// TIA Portal V18 export
FUNCTION "SS2_A3_32DI_IO_Update" : Void   // FC11140, LAD
{ S7_Optimized_Access := 'TRUE' }
VERSION : 0.1
// stored: AutoNumber false, IsIECCheckEnabled false, SetENOAutomatically false, UDAEnableTagReadback false
BEGIN

REGION Network 1: DIa0
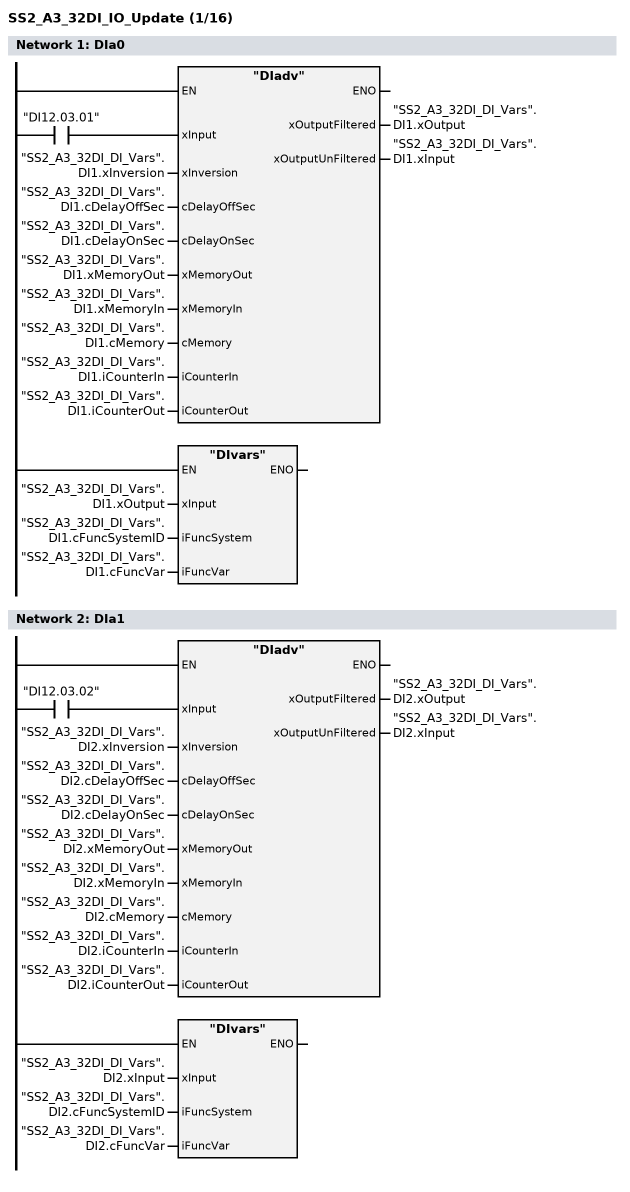
   RUNG wire#powerrail
      "DIadv"(xInput := wire#w1, xInversion := "SS2_A3_32DI_DI_Vars".DI1.xInversion, cDelayOffSec := "SS2_A3_32DI_DI_Vars".DI1.cDelayOffSec, cDelayOnSec := "SS2_A3_32DI_DI_Vars".DI1.cDelayOnSec, xMemoryOut := "SS2_A3_32DI_DI_Vars".DI1.xMemoryOut, xMemoryIn := "SS2_A3_32DI_DI_Vars".DI1.xMemoryIn, cMemory := "SS2_A3_32DI_DI_Vars".DI1.cMemory, iCounterIn := "SS2_A3_32DI_DI_Vars".DI1.iCounterIn, iCounterOut := "SS2_A3_32DI_DI_Vars".DI1.iCounterOut, xOutputFiltered => "SS2_A3_32DI_DI_Vars".DI1.xOutput, xOutputUnFiltered => "SS2_A3_32DI_DI_Vars".DI1.xInput)
   END_RUNG
   RUNG wire#powerrail
      Contact( "DI12.03.01" )
   END_RUNG wire#w1
   RUNG wire#powerrail
      "DIvars"(xInput := "SS2_A3_32DI_DI_Vars".DI1.xOutput, iFuncSystem := "SS2_A3_32DI_DI_Vars".DI1.cFuncSystemID, iFuncVar := "SS2_A3_32DI_DI_Vars".DI1.cFuncVar)
   END_RUNG
   // the same network as SCL:
   "DIadv"(xInput := "DI12.03.01",
           xInversion := "SS2_A3_32DI_DI_Vars".DI1.xInversion,
           cDelayOffSec := "SS2_A3_32DI_DI_Vars".DI1.cDelayOffSec,
           cDelayOnSec := "SS2_A3_32DI_DI_Vars".DI1.cDelayOnSec,
           xMemoryOut := "SS2_A3_32DI_DI_Vars".DI1.xMemoryOut,
           xMemoryIn := "SS2_A3_32DI_DI_Vars".DI1.xMemoryIn,
           cMemory := "SS2_A3_32DI_DI_Vars".DI1.cMemory,
           iCounterIn := "SS2_A3_32DI_DI_Vars".DI1.iCounterIn,
           iCounterOut := "SS2_A3_32DI_DI_Vars".DI1.iCounterOut,
           xOutputFiltered => "SS2_A3_32DI_DI_Vars".DI1.xOutput,
           xOutputUnFiltered => "SS2_A3_32DI_DI_Vars".DI1.xInput);
   "DIvars"(xInput := "SS2_A3_32DI_DI_Vars".DI1.xOutput,
            iFuncSystem := "SS2_A3_32DI_DI_Vars".DI1.cFuncSystemID,
            iFuncVar := "SS2_A3_32DI_DI_Vars".DI1.cFuncVar);
END_REGION

REGION Network 2: DIa1
   RUNG wire#powerrail
      "DIadv"(xInput := wire#w1, xInversion := "SS2_A3_32DI_DI_Vars".DI2.xInversion, cDelayOffSec := "SS2_A3_32DI_DI_Vars".DI2.cDelayOffSec, cDelayOnSec := "SS2_A3_32DI_DI_Vars".DI2.cDelayOnSec, xMemoryOut := "SS2_A3_32DI_DI_Vars".DI2.xMemoryOut, xMemoryIn := "SS2_A3_32DI_DI_Vars".DI2.xMemoryIn, cMemory := "SS2_A3_32DI_DI_Vars".DI2.cMemory, iCounterIn := "SS2_A3_32DI_DI_Vars".DI2.iCounterIn, iCounterOut := "SS2_A3_32DI_DI_Vars".DI2.iCounterOut, xOutputFiltered => "SS2_A3_32DI_DI_Vars".DI2.xOutput, xOutputUnFiltered => "SS2_A3_32DI_DI_Vars".DI2.xInput)
   END_RUNG
   RUNG wire#powerrail
      Contact( "DI12.03.02" )
   END_RUNG wire#w1
   RUNG wire#powerrail
      "DIvars"(xInput := "SS2_A3_32DI_DI_Vars".DI2.xInput, iFuncSystem := "SS2_A3_32DI_DI_Vars".DI2.cFuncSystemID, iFuncVar := "SS2_A3_32DI_DI_Vars".DI2.cFuncVar)
   END_RUNG
   // the same network as SCL:
   "DIadv"(xInput := "DI12.03.02",
           xInversion := "SS2_A3_32DI_DI_Vars".DI2.xInversion,
           cDelayOffSec := "SS2_A3_32DI_DI_Vars".DI2.cDelayOffSec,
           cDelayOnSec := "SS2_A3_32DI_DI_Vars".DI2.cDelayOnSec,
           xMemoryOut := "SS2_A3_32DI_DI_Vars".DI2.xMemoryOut,
           xMemoryIn := "SS2_A3_32DI_DI_Vars".DI2.xMemoryIn,
           cMemory := "SS2_A3_32DI_DI_Vars".DI2.cMemory,
           iCounterIn := "SS2_A3_32DI_DI_Vars".DI2.iCounterIn,
           iCounterOut := "SS2_A3_32DI_DI_Vars".DI2.iCounterOut,
           xOutputFiltered => "SS2_A3_32DI_DI_Vars".DI2.xOutput,
           xOutputUnFiltered => "SS2_A3_32DI_DI_Vars".DI2.xInput);
   "DIvars"(xInput := "SS2_A3_32DI_DI_Vars".DI2.xInput,
            iFuncSystem := "SS2_A3_32DI_DI_Vars".DI2.cFuncSystemID,
            iFuncVar := "SS2_A3_32DI_DI_Vars".DI2.cFuncVar);
END_REGION

REGION Network 3: DIa2
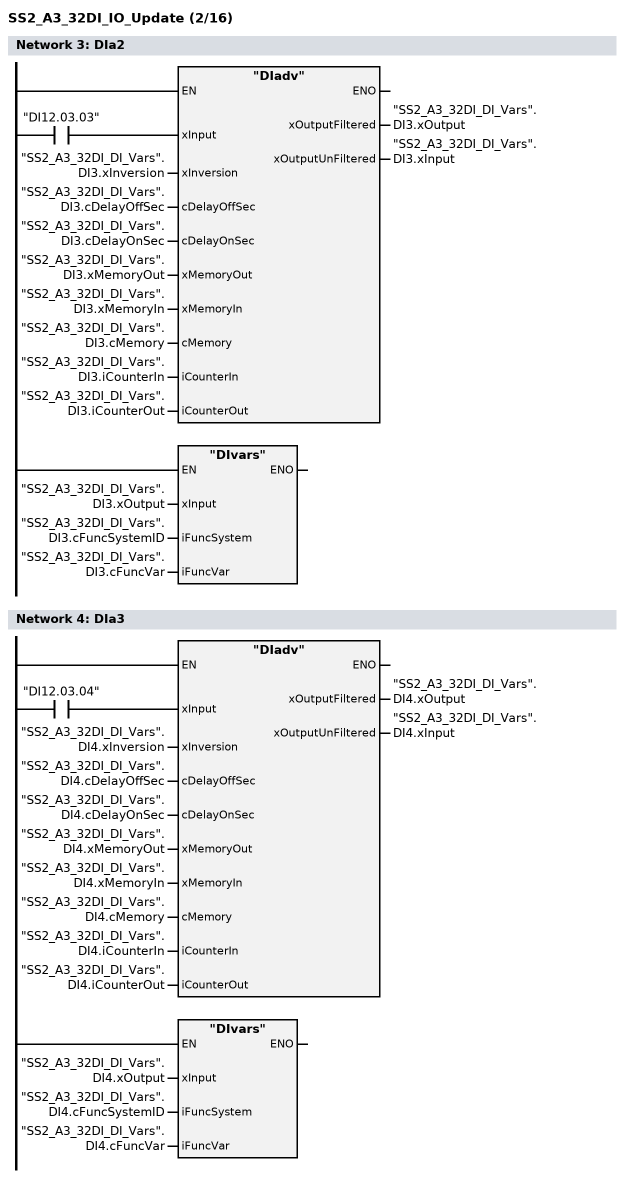
   RUNG wire#powerrail
      "DIadv"(xInput := wire#w1, xInversion := "SS2_A3_32DI_DI_Vars".DI3.xInversion, cDelayOffSec := "SS2_A3_32DI_DI_Vars".DI3.cDelayOffSec, cDelayOnSec := "SS2_A3_32DI_DI_Vars".DI3.cDelayOnSec, xMemoryOut := "SS2_A3_32DI_DI_Vars".DI3.xMemoryOut, xMemoryIn := "SS2_A3_32DI_DI_Vars".DI3.xMemoryIn, cMemory := "SS2_A3_32DI_DI_Vars".DI3.cMemory, iCounterIn := "SS2_A3_32DI_DI_Vars".DI3.iCounterIn, iCounterOut := "SS2_A3_32DI_DI_Vars".DI3.iCounterOut, xOutputFiltered => "SS2_A3_32DI_DI_Vars".DI3.xOutput, xOutputUnFiltered => "SS2_A3_32DI_DI_Vars".DI3.xInput)
   END_RUNG
   RUNG wire#powerrail
      Contact( "DI12.03.03" )
   END_RUNG wire#w1
   RUNG wire#powerrail
      "DIvars"(xInput := "SS2_A3_32DI_DI_Vars".DI3.xOutput, iFuncSystem := "SS2_A3_32DI_DI_Vars".DI3.cFuncSystemID, iFuncVar := "SS2_A3_32DI_DI_Vars".DI3.cFuncVar)
   END_RUNG
   // the same network as SCL:
   "DIadv"(xInput := "DI12.03.03",
           xInversion := "SS2_A3_32DI_DI_Vars".DI3.xInversion,
           cDelayOffSec := "SS2_A3_32DI_DI_Vars".DI3.cDelayOffSec,
           cDelayOnSec := "SS2_A3_32DI_DI_Vars".DI3.cDelayOnSec,
           xMemoryOut := "SS2_A3_32DI_DI_Vars".DI3.xMemoryOut,
           xMemoryIn := "SS2_A3_32DI_DI_Vars".DI3.xMemoryIn,
           cMemory := "SS2_A3_32DI_DI_Vars".DI3.cMemory,
           iCounterIn := "SS2_A3_32DI_DI_Vars".DI3.iCounterIn,
           iCounterOut := "SS2_A3_32DI_DI_Vars".DI3.iCounterOut,
           xOutputFiltered => "SS2_A3_32DI_DI_Vars".DI3.xOutput,
           xOutputUnFiltered => "SS2_A3_32DI_DI_Vars".DI3.xInput);
   "DIvars"(xInput := "SS2_A3_32DI_DI_Vars".DI3.xOutput,
            iFuncSystem := "SS2_A3_32DI_DI_Vars".DI3.cFuncSystemID,
            iFuncVar := "SS2_A3_32DI_DI_Vars".DI3.cFuncVar);
END_REGION

REGION Network 4: DIa3
   RUNG wire#powerrail
      "DIadv"(xInput := wire#w1, xInversion := "SS2_A3_32DI_DI_Vars".DI4.xInversion, cDelayOffSec := "SS2_A3_32DI_DI_Vars".DI4.cDelayOffSec, cDelayOnSec := "SS2_A3_32DI_DI_Vars".DI4.cDelayOnSec, xMemoryOut := "SS2_A3_32DI_DI_Vars".DI4.xMemoryOut, xMemoryIn := "SS2_A3_32DI_DI_Vars".DI4.xMemoryIn, cMemory := "SS2_A3_32DI_DI_Vars".DI4.cMemory, iCounterIn := "SS2_A3_32DI_DI_Vars".DI4.iCounterIn, iCounterOut := "SS2_A3_32DI_DI_Vars".DI4.iCounterOut, xOutputFiltered => "SS2_A3_32DI_DI_Vars".DI4.xOutput, xOutputUnFiltered => "SS2_A3_32DI_DI_Vars".DI4.xInput)
   END_RUNG
   RUNG wire#powerrail
      Contact( "DI12.03.04" )
   END_RUNG wire#w1
   RUNG wire#powerrail
      "DIvars"(xInput := "SS2_A3_32DI_DI_Vars".DI4.xOutput, iFuncSystem := "SS2_A3_32DI_DI_Vars".DI4.cFuncSystemID, iFuncVar := "SS2_A3_32DI_DI_Vars".DI4.cFuncVar)
   END_RUNG
   // the same network as SCL:
   "DIadv"(xInput := "DI12.03.04",
           xInversion := "SS2_A3_32DI_DI_Vars".DI4.xInversion,
           cDelayOffSec := "SS2_A3_32DI_DI_Vars".DI4.cDelayOffSec,
           cDelayOnSec := "SS2_A3_32DI_DI_Vars".DI4.cDelayOnSec,
           xMemoryOut := "SS2_A3_32DI_DI_Vars".DI4.xMemoryOut,
           xMemoryIn := "SS2_A3_32DI_DI_Vars".DI4.xMemoryIn,
           cMemory := "SS2_A3_32DI_DI_Vars".DI4.cMemory,
           iCounterIn := "SS2_A3_32DI_DI_Vars".DI4.iCounterIn,
           iCounterOut := "SS2_A3_32DI_DI_Vars".DI4.iCounterOut,
           xOutputFiltered => "SS2_A3_32DI_DI_Vars".DI4.xOutput,
           xOutputUnFiltered => "SS2_A3_32DI_DI_Vars".DI4.xInput);
   "DIvars"(xInput := "SS2_A3_32DI_DI_Vars".DI4.xOutput,
            iFuncSystem := "SS2_A3_32DI_DI_Vars".DI4.cFuncSystemID,
            iFuncVar := "SS2_A3_32DI_DI_Vars".DI4.cFuncVar);
END_REGION

REGION Network 5: DIa4
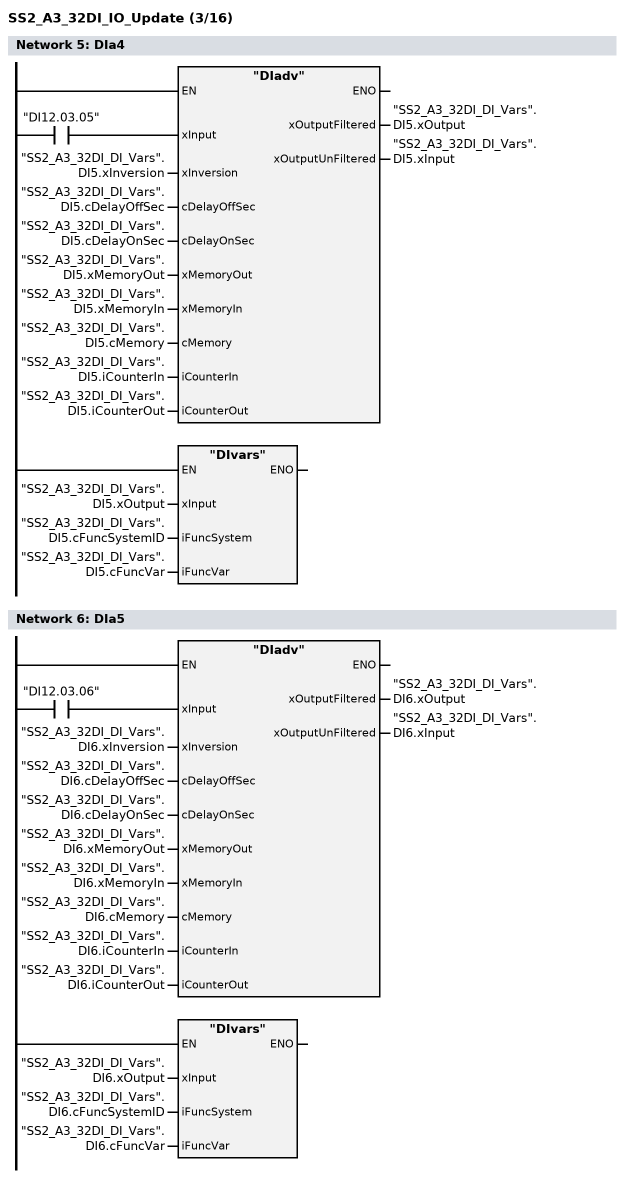
   RUNG wire#powerrail
      "DIadv"(xInput := wire#w1, xInversion := "SS2_A3_32DI_DI_Vars".DI5.xInversion, cDelayOffSec := "SS2_A3_32DI_DI_Vars".DI5.cDelayOffSec, cDelayOnSec := "SS2_A3_32DI_DI_Vars".DI5.cDelayOnSec, xMemoryOut := "SS2_A3_32DI_DI_Vars".DI5.xMemoryOut, xMemoryIn := "SS2_A3_32DI_DI_Vars".DI5.xMemoryIn, cMemory := "SS2_A3_32DI_DI_Vars".DI5.cMemory, iCounterIn := "SS2_A3_32DI_DI_Vars".DI5.iCounterIn, iCounterOut := "SS2_A3_32DI_DI_Vars".DI5.iCounterOut, xOutputFiltered => "SS2_A3_32DI_DI_Vars".DI5.xOutput, xOutputUnFiltered => "SS2_A3_32DI_DI_Vars".DI5.xInput)
   END_RUNG
   RUNG wire#powerrail
      Contact( "DI12.03.05" )
   END_RUNG wire#w1
   RUNG wire#powerrail
      "DIvars"(xInput := "SS2_A3_32DI_DI_Vars".DI5.xOutput, iFuncSystem := "SS2_A3_32DI_DI_Vars".DI5.cFuncSystemID, iFuncVar := "SS2_A3_32DI_DI_Vars".DI5.cFuncVar)
   END_RUNG
   // the same network as SCL:
   "DIadv"(xInput := "DI12.03.05",
           xInversion := "SS2_A3_32DI_DI_Vars".DI5.xInversion,
           cDelayOffSec := "SS2_A3_32DI_DI_Vars".DI5.cDelayOffSec,
           cDelayOnSec := "SS2_A3_32DI_DI_Vars".DI5.cDelayOnSec,
           xMemoryOut := "SS2_A3_32DI_DI_Vars".DI5.xMemoryOut,
           xMemoryIn := "SS2_A3_32DI_DI_Vars".DI5.xMemoryIn,
           cMemory := "SS2_A3_32DI_DI_Vars".DI5.cMemory,
           iCounterIn := "SS2_A3_32DI_DI_Vars".DI5.iCounterIn,
           iCounterOut := "SS2_A3_32DI_DI_Vars".DI5.iCounterOut,
           xOutputFiltered => "SS2_A3_32DI_DI_Vars".DI5.xOutput,
           xOutputUnFiltered => "SS2_A3_32DI_DI_Vars".DI5.xInput);
   "DIvars"(xInput := "SS2_A3_32DI_DI_Vars".DI5.xOutput,
            iFuncSystem := "SS2_A3_32DI_DI_Vars".DI5.cFuncSystemID,
            iFuncVar := "SS2_A3_32DI_DI_Vars".DI5.cFuncVar);
END_REGION

REGION Network 6: DIa5
   RUNG wire#powerrail
      "DIadv"(xInput := wire#w1, xInversion := "SS2_A3_32DI_DI_Vars".DI6.xInversion, cDelayOffSec := "SS2_A3_32DI_DI_Vars".DI6.cDelayOffSec, cDelayOnSec := "SS2_A3_32DI_DI_Vars".DI6.cDelayOnSec, xMemoryOut := "SS2_A3_32DI_DI_Vars".DI6.xMemoryOut, xMemoryIn := "SS2_A3_32DI_DI_Vars".DI6.xMemoryIn, cMemory := "SS2_A3_32DI_DI_Vars".DI6.cMemory, iCounterIn := "SS2_A3_32DI_DI_Vars".DI6.iCounterIn, iCounterOut := "SS2_A3_32DI_DI_Vars".DI6.iCounterOut, xOutputFiltered => "SS2_A3_32DI_DI_Vars".DI6.xOutput, xOutputUnFiltered => "SS2_A3_32DI_DI_Vars".DI6.xInput)
   END_RUNG
   RUNG wire#powerrail
      Contact( "DI12.03.06" )
   END_RUNG wire#w1
   RUNG wire#powerrail
      "DIvars"(xInput := "SS2_A3_32DI_DI_Vars".DI6.xOutput, iFuncSystem := "SS2_A3_32DI_DI_Vars".DI6.cFuncSystemID, iFuncVar := "SS2_A3_32DI_DI_Vars".DI6.cFuncVar)
   END_RUNG
   // the same network as SCL:
   "DIadv"(xInput := "DI12.03.06",
           xInversion := "SS2_A3_32DI_DI_Vars".DI6.xInversion,
           cDelayOffSec := "SS2_A3_32DI_DI_Vars".DI6.cDelayOffSec,
           cDelayOnSec := "SS2_A3_32DI_DI_Vars".DI6.cDelayOnSec,
           xMemoryOut := "SS2_A3_32DI_DI_Vars".DI6.xMemoryOut,
           xMemoryIn := "SS2_A3_32DI_DI_Vars".DI6.xMemoryIn,
           cMemory := "SS2_A3_32DI_DI_Vars".DI6.cMemory,
           iCounterIn := "SS2_A3_32DI_DI_Vars".DI6.iCounterIn,
           iCounterOut := "SS2_A3_32DI_DI_Vars".DI6.iCounterOut,
           xOutputFiltered => "SS2_A3_32DI_DI_Vars".DI6.xOutput,
           xOutputUnFiltered => "SS2_A3_32DI_DI_Vars".DI6.xInput);
   "DIvars"(xInput := "SS2_A3_32DI_DI_Vars".DI6.xOutput,
            iFuncSystem := "SS2_A3_32DI_DI_Vars".DI6.cFuncSystemID,
            iFuncVar := "SS2_A3_32DI_DI_Vars".DI6.cFuncVar);
END_REGION

REGION Network 7: DIa6
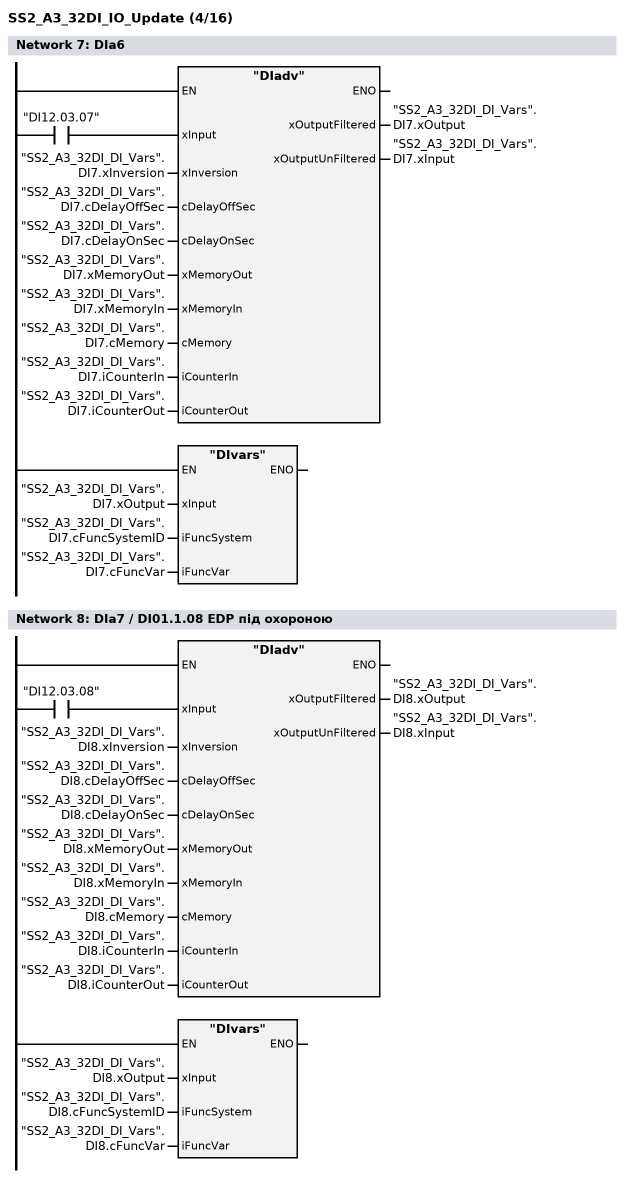
   RUNG wire#powerrail
      "DIadv"(xInput := wire#w1, xInversion := "SS2_A3_32DI_DI_Vars".DI7.xInversion, cDelayOffSec := "SS2_A3_32DI_DI_Vars".DI7.cDelayOffSec, cDelayOnSec := "SS2_A3_32DI_DI_Vars".DI7.cDelayOnSec, xMemoryOut := "SS2_A3_32DI_DI_Vars".DI7.xMemoryOut, xMemoryIn := "SS2_A3_32DI_DI_Vars".DI7.xMemoryIn, cMemory := "SS2_A3_32DI_DI_Vars".DI7.cMemory, iCounterIn := "SS2_A3_32DI_DI_Vars".DI7.iCounterIn, iCounterOut := "SS2_A3_32DI_DI_Vars".DI7.iCounterOut, xOutputFiltered => "SS2_A3_32DI_DI_Vars".DI7.xOutput, xOutputUnFiltered => "SS2_A3_32DI_DI_Vars".DI7.xInput)
   END_RUNG
   RUNG wire#powerrail
      Contact( "DI12.03.07" )
   END_RUNG wire#w1
   RUNG wire#powerrail
      "DIvars"(xInput := "SS2_A3_32DI_DI_Vars".DI7.xOutput, iFuncSystem := "SS2_A3_32DI_DI_Vars".DI7.cFuncSystemID, iFuncVar := "SS2_A3_32DI_DI_Vars".DI7.cFuncVar)
   END_RUNG
   // the same network as SCL:
   "DIadv"(xInput := "DI12.03.07",
           xInversion := "SS2_A3_32DI_DI_Vars".DI7.xInversion,
           cDelayOffSec := "SS2_A3_32DI_DI_Vars".DI7.cDelayOffSec,
           cDelayOnSec := "SS2_A3_32DI_DI_Vars".DI7.cDelayOnSec,
           xMemoryOut := "SS2_A3_32DI_DI_Vars".DI7.xMemoryOut,
           xMemoryIn := "SS2_A3_32DI_DI_Vars".DI7.xMemoryIn,
           cMemory := "SS2_A3_32DI_DI_Vars".DI7.cMemory,
           iCounterIn := "SS2_A3_32DI_DI_Vars".DI7.iCounterIn,
           iCounterOut := "SS2_A3_32DI_DI_Vars".DI7.iCounterOut,
           xOutputFiltered => "SS2_A3_32DI_DI_Vars".DI7.xOutput,
           xOutputUnFiltered => "SS2_A3_32DI_DI_Vars".DI7.xInput);
   "DIvars"(xInput := "SS2_A3_32DI_DI_Vars".DI7.xOutput,
            iFuncSystem := "SS2_A3_32DI_DI_Vars".DI7.cFuncSystemID,
            iFuncVar := "SS2_A3_32DI_DI_Vars".DI7.cFuncVar);
END_REGION

REGION Network 8: DIa7 / DI01.1.08 EDP під охороною
   RUNG wire#powerrail
      "DIadv"(xInput := wire#w1, xInversion := "SS2_A3_32DI_DI_Vars".DI8.xInversion, cDelayOffSec := "SS2_A3_32DI_DI_Vars".DI8.cDelayOffSec, cDelayOnSec := "SS2_A3_32DI_DI_Vars".DI8.cDelayOnSec, xMemoryOut := "SS2_A3_32DI_DI_Vars".DI8.xMemoryOut, xMemoryIn := "SS2_A3_32DI_DI_Vars".DI8.xMemoryIn, cMemory := "SS2_A3_32DI_DI_Vars".DI8.cMemory, iCounterIn := "SS2_A3_32DI_DI_Vars".DI8.iCounterIn, iCounterOut := "SS2_A3_32DI_DI_Vars".DI8.iCounterOut, xOutputFiltered => "SS2_A3_32DI_DI_Vars".DI8.xOutput, xOutputUnFiltered => "SS2_A3_32DI_DI_Vars".DI8.xInput)
   END_RUNG
   RUNG wire#powerrail
      Contact( "DI12.03.08" )
   END_RUNG wire#w1
   RUNG wire#powerrail
      "DIvars"(xInput := "SS2_A3_32DI_DI_Vars".DI8.xOutput, iFuncSystem := "SS2_A3_32DI_DI_Vars".DI8.cFuncSystemID, iFuncVar := "SS2_A3_32DI_DI_Vars".DI8.cFuncVar)
   END_RUNG
   // the same network as SCL:
   "DIadv"(xInput := "DI12.03.08",
           xInversion := "SS2_A3_32DI_DI_Vars".DI8.xInversion,
           cDelayOffSec := "SS2_A3_32DI_DI_Vars".DI8.cDelayOffSec,
           cDelayOnSec := "SS2_A3_32DI_DI_Vars".DI8.cDelayOnSec,
           xMemoryOut := "SS2_A3_32DI_DI_Vars".DI8.xMemoryOut,
           xMemoryIn := "SS2_A3_32DI_DI_Vars".DI8.xMemoryIn,
           cMemory := "SS2_A3_32DI_DI_Vars".DI8.cMemory,
           iCounterIn := "SS2_A3_32DI_DI_Vars".DI8.iCounterIn,
           iCounterOut := "SS2_A3_32DI_DI_Vars".DI8.iCounterOut,
           xOutputFiltered => "SS2_A3_32DI_DI_Vars".DI8.xOutput,
           xOutputUnFiltered => "SS2_A3_32DI_DI_Vars".DI8.xInput);
   "DIvars"(xInput := "SS2_A3_32DI_DI_Vars".DI8.xOutput,
            iFuncSystem := "SS2_A3_32DI_DI_Vars".DI8.cFuncSystemID,
            iFuncVar := "SS2_A3_32DI_DI_Vars".DI8.cFuncVar);
END_REGION

REGION Network 9: DIb0 / DI01.1.08 EDP під охороною
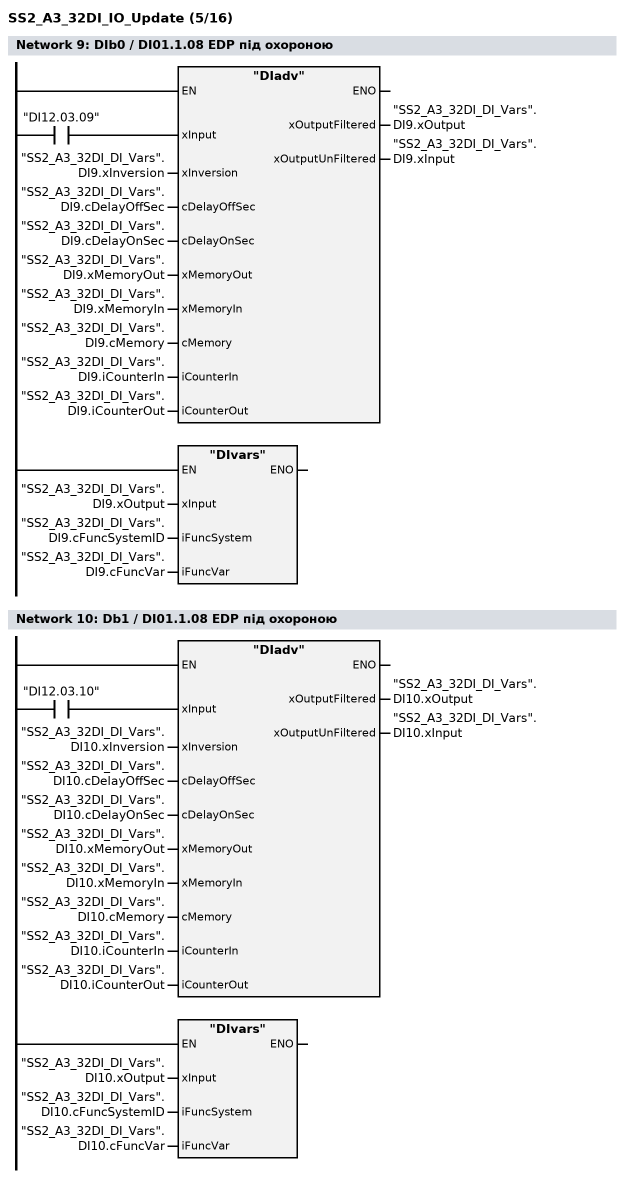
   RUNG wire#powerrail
      "DIadv"(xInput := wire#w1, xInversion := "SS2_A3_32DI_DI_Vars".DI9.xInversion, cDelayOffSec := "SS2_A3_32DI_DI_Vars".DI9.cDelayOffSec, cDelayOnSec := "SS2_A3_32DI_DI_Vars".DI9.cDelayOnSec, xMemoryOut := "SS2_A3_32DI_DI_Vars".DI9.xMemoryOut, xMemoryIn := "SS2_A3_32DI_DI_Vars".DI9.xMemoryIn, cMemory := "SS2_A3_32DI_DI_Vars".DI9.cMemory, iCounterIn := "SS2_A3_32DI_DI_Vars".DI9.iCounterIn, iCounterOut := "SS2_A3_32DI_DI_Vars".DI9.iCounterOut, xOutputFiltered => "SS2_A3_32DI_DI_Vars".DI9.xOutput, xOutputUnFiltered => "SS2_A3_32DI_DI_Vars".DI9.xInput)
   END_RUNG
   RUNG wire#powerrail
      Contact( "DI12.03.09" )
   END_RUNG wire#w1
   RUNG wire#powerrail
      "DIvars"(xInput := "SS2_A3_32DI_DI_Vars".DI9.xOutput, iFuncSystem := "SS2_A3_32DI_DI_Vars".DI9.cFuncSystemID, iFuncVar := "SS2_A3_32DI_DI_Vars".DI9.cFuncVar)
   END_RUNG
   // the same network as SCL:
   "DIadv"(xInput := "DI12.03.09",
           xInversion := "SS2_A3_32DI_DI_Vars".DI9.xInversion,
           cDelayOffSec := "SS2_A3_32DI_DI_Vars".DI9.cDelayOffSec,
           cDelayOnSec := "SS2_A3_32DI_DI_Vars".DI9.cDelayOnSec,
           xMemoryOut := "SS2_A3_32DI_DI_Vars".DI9.xMemoryOut,
           xMemoryIn := "SS2_A3_32DI_DI_Vars".DI9.xMemoryIn,
           cMemory := "SS2_A3_32DI_DI_Vars".DI9.cMemory,
           iCounterIn := "SS2_A3_32DI_DI_Vars".DI9.iCounterIn,
           iCounterOut := "SS2_A3_32DI_DI_Vars".DI9.iCounterOut,
           xOutputFiltered => "SS2_A3_32DI_DI_Vars".DI9.xOutput,
           xOutputUnFiltered => "SS2_A3_32DI_DI_Vars".DI9.xInput);
   "DIvars"(xInput := "SS2_A3_32DI_DI_Vars".DI9.xOutput,
            iFuncSystem := "SS2_A3_32DI_DI_Vars".DI9.cFuncSystemID,
            iFuncVar := "SS2_A3_32DI_DI_Vars".DI9.cFuncVar);
END_REGION

REGION Network 10: Db1 / DI01.1.08 EDP під охороною
   RUNG wire#powerrail
      "DIadv"(xInput := wire#w1, xInversion := "SS2_A3_32DI_DI_Vars".DI10.xInversion, cDelayOffSec := "SS2_A3_32DI_DI_Vars".DI10.cDelayOffSec, cDelayOnSec := "SS2_A3_32DI_DI_Vars".DI10.cDelayOnSec, xMemoryOut := "SS2_A3_32DI_DI_Vars".DI10.xMemoryOut, xMemoryIn := "SS2_A3_32DI_DI_Vars".DI10.xMemoryIn, cMemory := "SS2_A3_32DI_DI_Vars".DI10.cMemory, iCounterIn := "SS2_A3_32DI_DI_Vars".DI10.iCounterIn, iCounterOut := "SS2_A3_32DI_DI_Vars".DI10.iCounterOut, xOutputFiltered => "SS2_A3_32DI_DI_Vars".DI10.xOutput, xOutputUnFiltered => "SS2_A3_32DI_DI_Vars".DI10.xInput)
   END_RUNG
   RUNG wire#powerrail
      Contact( "DI12.03.10" )
   END_RUNG wire#w1
   RUNG wire#powerrail
      "DIvars"(xInput := "SS2_A3_32DI_DI_Vars".DI10.xOutput, iFuncSystem := "SS2_A3_32DI_DI_Vars".DI10.cFuncSystemID, iFuncVar := "SS2_A3_32DI_DI_Vars".DI10.cFuncVar)
   END_RUNG
   // the same network as SCL:
   "DIadv"(xInput := "DI12.03.10",
           xInversion := "SS2_A3_32DI_DI_Vars".DI10.xInversion,
           cDelayOffSec := "SS2_A3_32DI_DI_Vars".DI10.cDelayOffSec,
           cDelayOnSec := "SS2_A3_32DI_DI_Vars".DI10.cDelayOnSec,
           xMemoryOut := "SS2_A3_32DI_DI_Vars".DI10.xMemoryOut,
           xMemoryIn := "SS2_A3_32DI_DI_Vars".DI10.xMemoryIn,
           cMemory := "SS2_A3_32DI_DI_Vars".DI10.cMemory,
           iCounterIn := "SS2_A3_32DI_DI_Vars".DI10.iCounterIn,
           iCounterOut := "SS2_A3_32DI_DI_Vars".DI10.iCounterOut,
           xOutputFiltered => "SS2_A3_32DI_DI_Vars".DI10.xOutput,
           xOutputUnFiltered => "SS2_A3_32DI_DI_Vars".DI10.xInput);
   "DIvars"(xInput := "SS2_A3_32DI_DI_Vars".DI10.xOutput,
            iFuncSystem := "SS2_A3_32DI_DI_Vars".DI10.cFuncSystemID,
            iFuncVar := "SS2_A3_32DI_DI_Vars".DI10.cFuncVar);
END_REGION

REGION Network 11: DIb2 / DI01.1.08 EDP під охороною
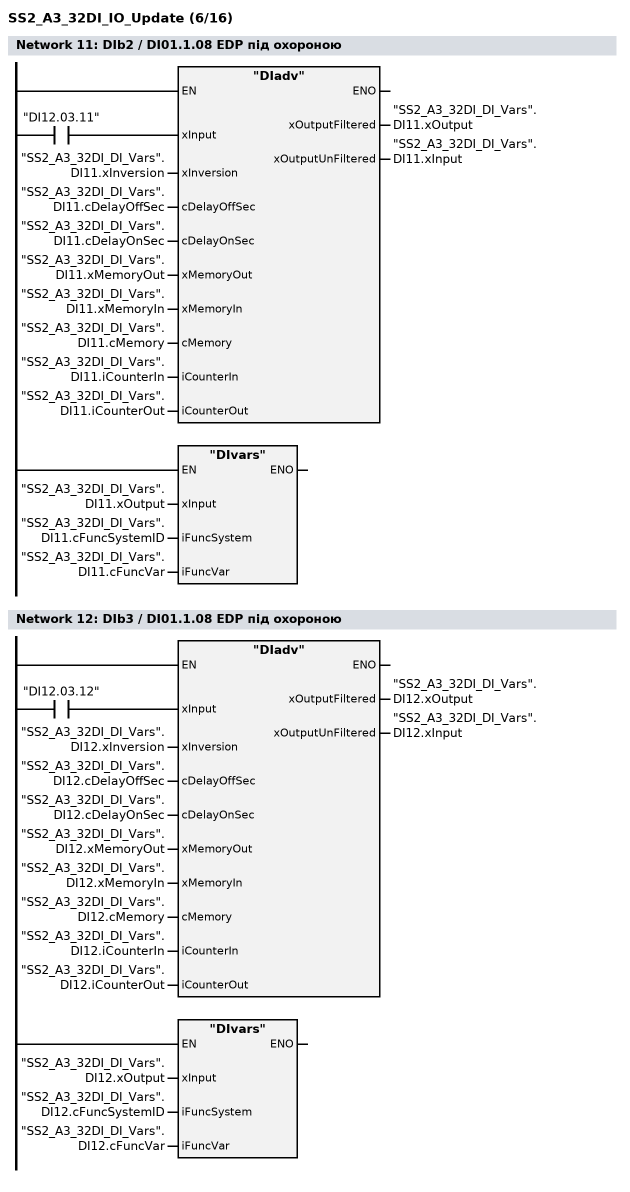
   RUNG wire#powerrail
      "DIadv"(xInput := wire#w1, xInversion := "SS2_A3_32DI_DI_Vars".DI11.xInversion, cDelayOffSec := "SS2_A3_32DI_DI_Vars".DI11.cDelayOffSec, cDelayOnSec := "SS2_A3_32DI_DI_Vars".DI11.cDelayOnSec, xMemoryOut := "SS2_A3_32DI_DI_Vars".DI11.xMemoryOut, xMemoryIn := "SS2_A3_32DI_DI_Vars".DI11.xMemoryIn, cMemory := "SS2_A3_32DI_DI_Vars".DI11.cMemory, iCounterIn := "SS2_A3_32DI_DI_Vars".DI11.iCounterIn, iCounterOut := "SS2_A3_32DI_DI_Vars".DI11.iCounterOut, xOutputFiltered => "SS2_A3_32DI_DI_Vars".DI11.xOutput, xOutputUnFiltered => "SS2_A3_32DI_DI_Vars".DI11.xInput)
   END_RUNG
   RUNG wire#powerrail
      Contact( "DI12.03.11" )
   END_RUNG wire#w1
   RUNG wire#powerrail
      "DIvars"(xInput := "SS2_A3_32DI_DI_Vars".DI11.xOutput, iFuncSystem := "SS2_A3_32DI_DI_Vars".DI11.cFuncSystemID, iFuncVar := "SS2_A3_32DI_DI_Vars".DI11.cFuncVar)
   END_RUNG
   // the same network as SCL:
   "DIadv"(xInput := "DI12.03.11",
           xInversion := "SS2_A3_32DI_DI_Vars".DI11.xInversion,
           cDelayOffSec := "SS2_A3_32DI_DI_Vars".DI11.cDelayOffSec,
           cDelayOnSec := "SS2_A3_32DI_DI_Vars".DI11.cDelayOnSec,
           xMemoryOut := "SS2_A3_32DI_DI_Vars".DI11.xMemoryOut,
           xMemoryIn := "SS2_A3_32DI_DI_Vars".DI11.xMemoryIn,
           cMemory := "SS2_A3_32DI_DI_Vars".DI11.cMemory,
           iCounterIn := "SS2_A3_32DI_DI_Vars".DI11.iCounterIn,
           iCounterOut := "SS2_A3_32DI_DI_Vars".DI11.iCounterOut,
           xOutputFiltered => "SS2_A3_32DI_DI_Vars".DI11.xOutput,
           xOutputUnFiltered => "SS2_A3_32DI_DI_Vars".DI11.xInput);
   "DIvars"(xInput := "SS2_A3_32DI_DI_Vars".DI11.xOutput,
            iFuncSystem := "SS2_A3_32DI_DI_Vars".DI11.cFuncSystemID,
            iFuncVar := "SS2_A3_32DI_DI_Vars".DI11.cFuncVar);
END_REGION

REGION Network 12: DIb3 / DI01.1.08 EDP під охороною
   RUNG wire#powerrail
      "DIadv"(xInput := wire#w1, xInversion := "SS2_A3_32DI_DI_Vars".DI12.xInversion, cDelayOffSec := "SS2_A3_32DI_DI_Vars".DI12.cDelayOffSec, cDelayOnSec := "SS2_A3_32DI_DI_Vars".DI12.cDelayOnSec, xMemoryOut := "SS2_A3_32DI_DI_Vars".DI12.xMemoryOut, xMemoryIn := "SS2_A3_32DI_DI_Vars".DI12.xMemoryIn, cMemory := "SS2_A3_32DI_DI_Vars".DI12.cMemory, iCounterIn := "SS2_A3_32DI_DI_Vars".DI12.iCounterIn, iCounterOut := "SS2_A3_32DI_DI_Vars".DI12.iCounterOut, xOutputFiltered => "SS2_A3_32DI_DI_Vars".DI12.xOutput, xOutputUnFiltered => "SS2_A3_32DI_DI_Vars".DI12.xInput)
   END_RUNG
   RUNG wire#powerrail
      Contact( "DI12.03.12" )
   END_RUNG wire#w1
   RUNG wire#powerrail
      "DIvars"(xInput := "SS2_A3_32DI_DI_Vars".DI12.xOutput, iFuncSystem := "SS2_A3_32DI_DI_Vars".DI12.cFuncSystemID, iFuncVar := "SS2_A3_32DI_DI_Vars".DI12.cFuncVar)
   END_RUNG
   // the same network as SCL:
   "DIadv"(xInput := "DI12.03.12",
           xInversion := "SS2_A3_32DI_DI_Vars".DI12.xInversion,
           cDelayOffSec := "SS2_A3_32DI_DI_Vars".DI12.cDelayOffSec,
           cDelayOnSec := "SS2_A3_32DI_DI_Vars".DI12.cDelayOnSec,
           xMemoryOut := "SS2_A3_32DI_DI_Vars".DI12.xMemoryOut,
           xMemoryIn := "SS2_A3_32DI_DI_Vars".DI12.xMemoryIn,
           cMemory := "SS2_A3_32DI_DI_Vars".DI12.cMemory,
           iCounterIn := "SS2_A3_32DI_DI_Vars".DI12.iCounterIn,
           iCounterOut := "SS2_A3_32DI_DI_Vars".DI12.iCounterOut,
           xOutputFiltered => "SS2_A3_32DI_DI_Vars".DI12.xOutput,
           xOutputUnFiltered => "SS2_A3_32DI_DI_Vars".DI12.xInput);
   "DIvars"(xInput := "SS2_A3_32DI_DI_Vars".DI12.xOutput,
            iFuncSystem := "SS2_A3_32DI_DI_Vars".DI12.cFuncSystemID,
            iFuncVar := "SS2_A3_32DI_DI_Vars".DI12.cFuncVar);
END_REGION

REGION Network 13: DIb4 / DI01.1.08 EDP під охороною
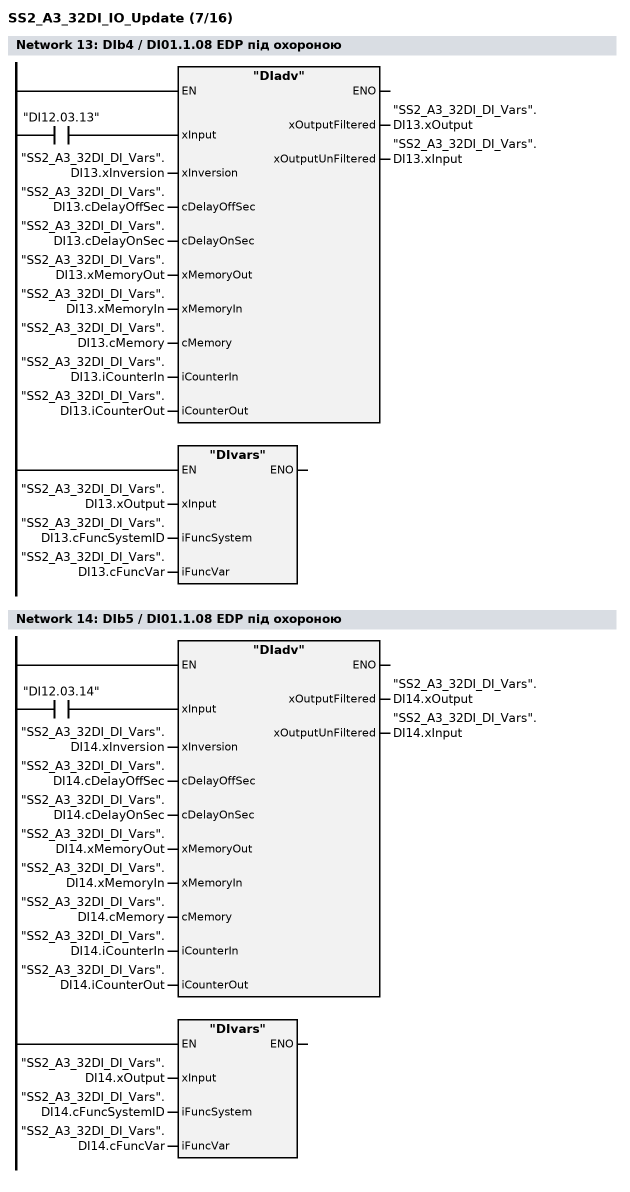
   RUNG wire#powerrail
      "DIadv"(xInput := wire#w1, xInversion := "SS2_A3_32DI_DI_Vars".DI13.xInversion, cDelayOffSec := "SS2_A3_32DI_DI_Vars".DI13.cDelayOffSec, cDelayOnSec := "SS2_A3_32DI_DI_Vars".DI13.cDelayOnSec, xMemoryOut := "SS2_A3_32DI_DI_Vars".DI13.xMemoryOut, xMemoryIn := "SS2_A3_32DI_DI_Vars".DI13.xMemoryIn, cMemory := "SS2_A3_32DI_DI_Vars".DI13.cMemory, iCounterIn := "SS2_A3_32DI_DI_Vars".DI13.iCounterIn, iCounterOut := "SS2_A3_32DI_DI_Vars".DI13.iCounterOut, xOutputFiltered => "SS2_A3_32DI_DI_Vars".DI13.xOutput, xOutputUnFiltered => "SS2_A3_32DI_DI_Vars".DI13.xInput)
   END_RUNG
   RUNG wire#powerrail
      Contact( "DI12.03.13" )
   END_RUNG wire#w1
   RUNG wire#powerrail
      "DIvars"(xInput := "SS2_A3_32DI_DI_Vars".DI13.xOutput, iFuncSystem := "SS2_A3_32DI_DI_Vars".DI13.cFuncSystemID, iFuncVar := "SS2_A3_32DI_DI_Vars".DI13.cFuncVar)
   END_RUNG
   // the same network as SCL:
   "DIadv"(xInput := "DI12.03.13",
           xInversion := "SS2_A3_32DI_DI_Vars".DI13.xInversion,
           cDelayOffSec := "SS2_A3_32DI_DI_Vars".DI13.cDelayOffSec,
           cDelayOnSec := "SS2_A3_32DI_DI_Vars".DI13.cDelayOnSec,
           xMemoryOut := "SS2_A3_32DI_DI_Vars".DI13.xMemoryOut,
           xMemoryIn := "SS2_A3_32DI_DI_Vars".DI13.xMemoryIn,
           cMemory := "SS2_A3_32DI_DI_Vars".DI13.cMemory,
           iCounterIn := "SS2_A3_32DI_DI_Vars".DI13.iCounterIn,
           iCounterOut := "SS2_A3_32DI_DI_Vars".DI13.iCounterOut,
           xOutputFiltered => "SS2_A3_32DI_DI_Vars".DI13.xOutput,
           xOutputUnFiltered => "SS2_A3_32DI_DI_Vars".DI13.xInput);
   "DIvars"(xInput := "SS2_A3_32DI_DI_Vars".DI13.xOutput,
            iFuncSystem := "SS2_A3_32DI_DI_Vars".DI13.cFuncSystemID,
            iFuncVar := "SS2_A3_32DI_DI_Vars".DI13.cFuncVar);
END_REGION

REGION Network 14: DIb5 / DI01.1.08 EDP під охороною
   RUNG wire#powerrail
      "DIadv"(xInput := wire#w1, xInversion := "SS2_A3_32DI_DI_Vars".DI14.xInversion, cDelayOffSec := "SS2_A3_32DI_DI_Vars".DI14.cDelayOffSec, cDelayOnSec := "SS2_A3_32DI_DI_Vars".DI14.cDelayOnSec, xMemoryOut := "SS2_A3_32DI_DI_Vars".DI14.xMemoryOut, xMemoryIn := "SS2_A3_32DI_DI_Vars".DI14.xMemoryIn, cMemory := "SS2_A3_32DI_DI_Vars".DI14.cMemory, iCounterIn := "SS2_A3_32DI_DI_Vars".DI14.iCounterIn, iCounterOut := "SS2_A3_32DI_DI_Vars".DI14.iCounterOut, xOutputFiltered => "SS2_A3_32DI_DI_Vars".DI14.xOutput, xOutputUnFiltered => "SS2_A3_32DI_DI_Vars".DI14.xInput)
   END_RUNG
   RUNG wire#powerrail
      Contact( "DI12.03.14" )
   END_RUNG wire#w1
   RUNG wire#powerrail
      "DIvars"(xInput := "SS2_A3_32DI_DI_Vars".DI14.xOutput, iFuncSystem := "SS2_A3_32DI_DI_Vars".DI14.cFuncSystemID, iFuncVar := "SS2_A3_32DI_DI_Vars".DI14.cFuncVar)
   END_RUNG
   // the same network as SCL:
   "DIadv"(xInput := "DI12.03.14",
           xInversion := "SS2_A3_32DI_DI_Vars".DI14.xInversion,
           cDelayOffSec := "SS2_A3_32DI_DI_Vars".DI14.cDelayOffSec,
           cDelayOnSec := "SS2_A3_32DI_DI_Vars".DI14.cDelayOnSec,
           xMemoryOut := "SS2_A3_32DI_DI_Vars".DI14.xMemoryOut,
           xMemoryIn := "SS2_A3_32DI_DI_Vars".DI14.xMemoryIn,
           cMemory := "SS2_A3_32DI_DI_Vars".DI14.cMemory,
           iCounterIn := "SS2_A3_32DI_DI_Vars".DI14.iCounterIn,
           iCounterOut := "SS2_A3_32DI_DI_Vars".DI14.iCounterOut,
           xOutputFiltered => "SS2_A3_32DI_DI_Vars".DI14.xOutput,
           xOutputUnFiltered => "SS2_A3_32DI_DI_Vars".DI14.xInput);
   "DIvars"(xInput := "SS2_A3_32DI_DI_Vars".DI14.xOutput,
            iFuncSystem := "SS2_A3_32DI_DI_Vars".DI14.cFuncSystemID,
            iFuncVar := "SS2_A3_32DI_DI_Vars".DI14.cFuncVar);
END_REGION

REGION Network 15: DIb6 / DI01.1.08 EDP під охороною
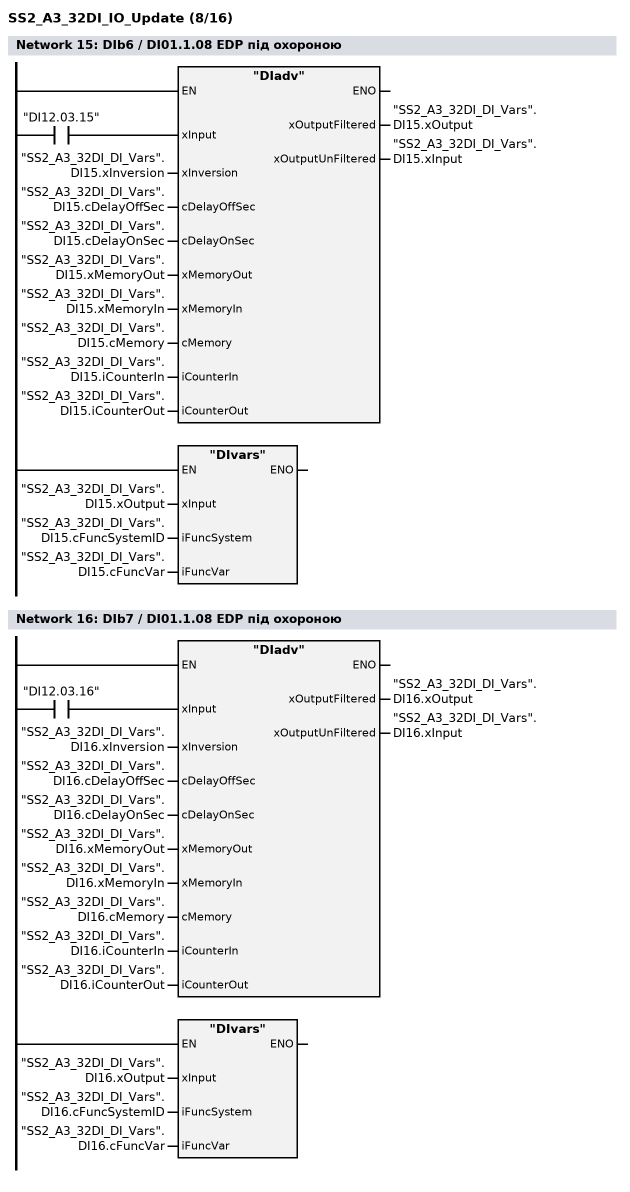
   RUNG wire#powerrail
      "DIadv"(xInput := wire#w1, xInversion := "SS2_A3_32DI_DI_Vars".DI15.xInversion, cDelayOffSec := "SS2_A3_32DI_DI_Vars".DI15.cDelayOffSec, cDelayOnSec := "SS2_A3_32DI_DI_Vars".DI15.cDelayOnSec, xMemoryOut := "SS2_A3_32DI_DI_Vars".DI15.xMemoryOut, xMemoryIn := "SS2_A3_32DI_DI_Vars".DI15.xMemoryIn, cMemory := "SS2_A3_32DI_DI_Vars".DI15.cMemory, iCounterIn := "SS2_A3_32DI_DI_Vars".DI15.iCounterIn, iCounterOut := "SS2_A3_32DI_DI_Vars".DI15.iCounterOut, xOutputFiltered => "SS2_A3_32DI_DI_Vars".DI15.xOutput, xOutputUnFiltered => "SS2_A3_32DI_DI_Vars".DI15.xInput)
   END_RUNG
   RUNG wire#powerrail
      Contact( "DI12.03.15" )
   END_RUNG wire#w1
   RUNG wire#powerrail
      "DIvars"(xInput := "SS2_A3_32DI_DI_Vars".DI15.xOutput, iFuncSystem := "SS2_A3_32DI_DI_Vars".DI15.cFuncSystemID, iFuncVar := "SS2_A3_32DI_DI_Vars".DI15.cFuncVar)
   END_RUNG
   // the same network as SCL:
   "DIadv"(xInput := "DI12.03.15",
           xInversion := "SS2_A3_32DI_DI_Vars".DI15.xInversion,
           cDelayOffSec := "SS2_A3_32DI_DI_Vars".DI15.cDelayOffSec,
           cDelayOnSec := "SS2_A3_32DI_DI_Vars".DI15.cDelayOnSec,
           xMemoryOut := "SS2_A3_32DI_DI_Vars".DI15.xMemoryOut,
           xMemoryIn := "SS2_A3_32DI_DI_Vars".DI15.xMemoryIn,
           cMemory := "SS2_A3_32DI_DI_Vars".DI15.cMemory,
           iCounterIn := "SS2_A3_32DI_DI_Vars".DI15.iCounterIn,
           iCounterOut := "SS2_A3_32DI_DI_Vars".DI15.iCounterOut,
           xOutputFiltered => "SS2_A3_32DI_DI_Vars".DI15.xOutput,
           xOutputUnFiltered => "SS2_A3_32DI_DI_Vars".DI15.xInput);
   "DIvars"(xInput := "SS2_A3_32DI_DI_Vars".DI15.xOutput,
            iFuncSystem := "SS2_A3_32DI_DI_Vars".DI15.cFuncSystemID,
            iFuncVar := "SS2_A3_32DI_DI_Vars".DI15.cFuncVar);
END_REGION

REGION Network 16: DIb7 / DI01.1.08 EDP під охороною
   RUNG wire#powerrail
      "DIadv"(xInput := wire#w1, xInversion := "SS2_A3_32DI_DI_Vars".DI16.xInversion, cDelayOffSec := "SS2_A3_32DI_DI_Vars".DI16.cDelayOffSec, cDelayOnSec := "SS2_A3_32DI_DI_Vars".DI16.cDelayOnSec, xMemoryOut := "SS2_A3_32DI_DI_Vars".DI16.xMemoryOut, xMemoryIn := "SS2_A3_32DI_DI_Vars".DI16.xMemoryIn, cMemory := "SS2_A3_32DI_DI_Vars".DI16.cMemory, iCounterIn := "SS2_A3_32DI_DI_Vars".DI16.iCounterIn, iCounterOut := "SS2_A3_32DI_DI_Vars".DI16.iCounterOut, xOutputFiltered => "SS2_A3_32DI_DI_Vars".DI16.xOutput, xOutputUnFiltered => "SS2_A3_32DI_DI_Vars".DI16.xInput)
   END_RUNG
   RUNG wire#powerrail
      Contact( "DI12.03.16" )
   END_RUNG wire#w1
   RUNG wire#powerrail
      "DIvars"(xInput := "SS2_A3_32DI_DI_Vars".DI16.xOutput, iFuncSystem := "SS2_A3_32DI_DI_Vars".DI16.cFuncSystemID, iFuncVar := "SS2_A3_32DI_DI_Vars".DI16.cFuncVar)
   END_RUNG
   // the same network as SCL:
   "DIadv"(xInput := "DI12.03.16",
           xInversion := "SS2_A3_32DI_DI_Vars".DI16.xInversion,
           cDelayOffSec := "SS2_A3_32DI_DI_Vars".DI16.cDelayOffSec,
           cDelayOnSec := "SS2_A3_32DI_DI_Vars".DI16.cDelayOnSec,
           xMemoryOut := "SS2_A3_32DI_DI_Vars".DI16.xMemoryOut,
           xMemoryIn := "SS2_A3_32DI_DI_Vars".DI16.xMemoryIn,
           cMemory := "SS2_A3_32DI_DI_Vars".DI16.cMemory,
           iCounterIn := "SS2_A3_32DI_DI_Vars".DI16.iCounterIn,
           iCounterOut := "SS2_A3_32DI_DI_Vars".DI16.iCounterOut,
           xOutputFiltered => "SS2_A3_32DI_DI_Vars".DI16.xOutput,
           xOutputUnFiltered => "SS2_A3_32DI_DI_Vars".DI16.xInput);
   "DIvars"(xInput := "SS2_A3_32DI_DI_Vars".DI16.xOutput,
            iFuncSystem := "SS2_A3_32DI_DI_Vars".DI16.cFuncSystemID,
            iFuncVar := "SS2_A3_32DI_DI_Vars".DI16.cFuncVar);
END_REGION

REGION Network 17: DIc0 / DI01.1.08 EDP під охороною
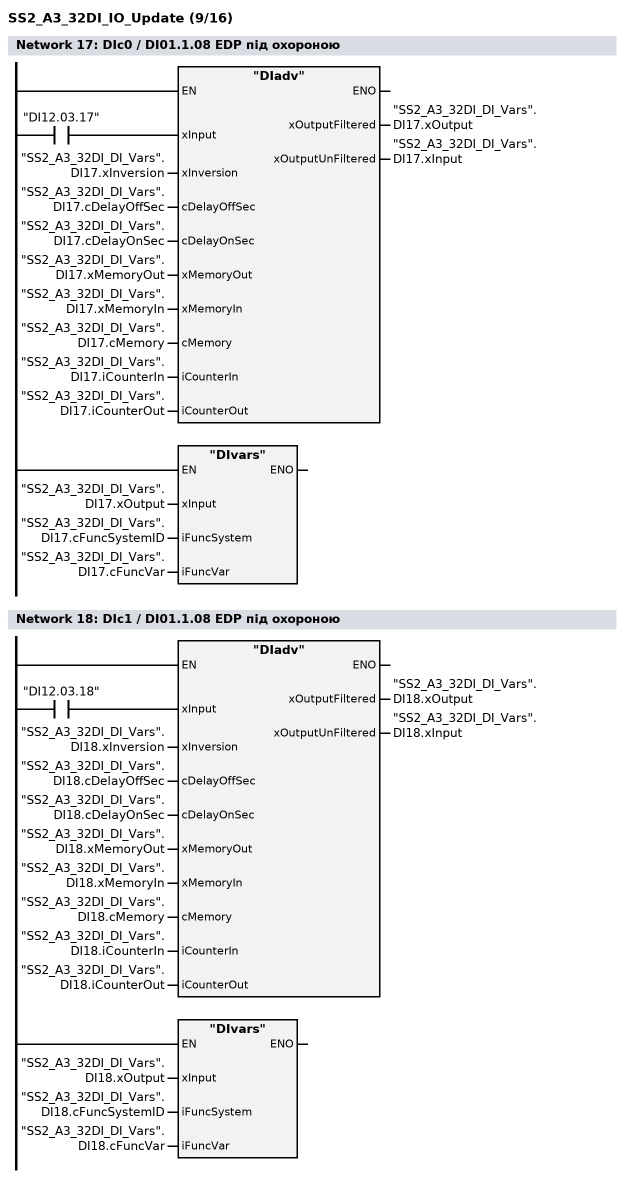
   RUNG wire#powerrail
      "DIadv"(xInput := wire#w1, xInversion := "SS2_A3_32DI_DI_Vars".DI17.xInversion, cDelayOffSec := "SS2_A3_32DI_DI_Vars".DI17.cDelayOffSec, cDelayOnSec := "SS2_A3_32DI_DI_Vars".DI17.cDelayOnSec, xMemoryOut := "SS2_A3_32DI_DI_Vars".DI17.xMemoryOut, xMemoryIn := "SS2_A3_32DI_DI_Vars".DI17.xMemoryIn, cMemory := "SS2_A3_32DI_DI_Vars".DI17.cMemory, iCounterIn := "SS2_A3_32DI_DI_Vars".DI17.iCounterIn, iCounterOut := "SS2_A3_32DI_DI_Vars".DI17.iCounterOut, xOutputFiltered => "SS2_A3_32DI_DI_Vars".DI17.xOutput, xOutputUnFiltered => "SS2_A3_32DI_DI_Vars".DI17.xInput)
   END_RUNG
   RUNG wire#powerrail
      Contact( "DI12.03.17" )
   END_RUNG wire#w1
   RUNG wire#powerrail
      "DIvars"(xInput := "SS2_A3_32DI_DI_Vars".DI17.xOutput, iFuncSystem := "SS2_A3_32DI_DI_Vars".DI17.cFuncSystemID, iFuncVar := "SS2_A3_32DI_DI_Vars".DI17.cFuncVar)
   END_RUNG
   // the same network as SCL:
   "DIadv"(xInput := "DI12.03.17",
           xInversion := "SS2_A3_32DI_DI_Vars".DI17.xInversion,
           cDelayOffSec := "SS2_A3_32DI_DI_Vars".DI17.cDelayOffSec,
           cDelayOnSec := "SS2_A3_32DI_DI_Vars".DI17.cDelayOnSec,
           xMemoryOut := "SS2_A3_32DI_DI_Vars".DI17.xMemoryOut,
           xMemoryIn := "SS2_A3_32DI_DI_Vars".DI17.xMemoryIn,
           cMemory := "SS2_A3_32DI_DI_Vars".DI17.cMemory,
           iCounterIn := "SS2_A3_32DI_DI_Vars".DI17.iCounterIn,
           iCounterOut := "SS2_A3_32DI_DI_Vars".DI17.iCounterOut,
           xOutputFiltered => "SS2_A3_32DI_DI_Vars".DI17.xOutput,
           xOutputUnFiltered => "SS2_A3_32DI_DI_Vars".DI17.xInput);
   "DIvars"(xInput := "SS2_A3_32DI_DI_Vars".DI17.xOutput,
            iFuncSystem := "SS2_A3_32DI_DI_Vars".DI17.cFuncSystemID,
            iFuncVar := "SS2_A3_32DI_DI_Vars".DI17.cFuncVar);
END_REGION

REGION Network 18: DIc1 / DI01.1.08 EDP під охороною
   RUNG wire#powerrail
      "DIadv"(xInput := wire#w1, xInversion := "SS2_A3_32DI_DI_Vars".DI18.xInversion, cDelayOffSec := "SS2_A3_32DI_DI_Vars".DI18.cDelayOffSec, cDelayOnSec := "SS2_A3_32DI_DI_Vars".DI18.cDelayOnSec, xMemoryOut := "SS2_A3_32DI_DI_Vars".DI18.xMemoryOut, xMemoryIn := "SS2_A3_32DI_DI_Vars".DI18.xMemoryIn, cMemory := "SS2_A3_32DI_DI_Vars".DI18.cMemory, iCounterIn := "SS2_A3_32DI_DI_Vars".DI18.iCounterIn, iCounterOut := "SS2_A3_32DI_DI_Vars".DI18.iCounterOut, xOutputFiltered => "SS2_A3_32DI_DI_Vars".DI18.xOutput, xOutputUnFiltered => "SS2_A3_32DI_DI_Vars".DI18.xInput)
   END_RUNG
   RUNG wire#powerrail
      Contact( "DI12.03.18" )
   END_RUNG wire#w1
   RUNG wire#powerrail
      "DIvars"(xInput := "SS2_A3_32DI_DI_Vars".DI18.xOutput, iFuncSystem := "SS2_A3_32DI_DI_Vars".DI18.cFuncSystemID, iFuncVar := "SS2_A3_32DI_DI_Vars".DI18.cFuncVar)
   END_RUNG
   // the same network as SCL:
   "DIadv"(xInput := "DI12.03.18",
           xInversion := "SS2_A3_32DI_DI_Vars".DI18.xInversion,
           cDelayOffSec := "SS2_A3_32DI_DI_Vars".DI18.cDelayOffSec,
           cDelayOnSec := "SS2_A3_32DI_DI_Vars".DI18.cDelayOnSec,
           xMemoryOut := "SS2_A3_32DI_DI_Vars".DI18.xMemoryOut,
           xMemoryIn := "SS2_A3_32DI_DI_Vars".DI18.xMemoryIn,
           cMemory := "SS2_A3_32DI_DI_Vars".DI18.cMemory,
           iCounterIn := "SS2_A3_32DI_DI_Vars".DI18.iCounterIn,
           iCounterOut := "SS2_A3_32DI_DI_Vars".DI18.iCounterOut,
           xOutputFiltered => "SS2_A3_32DI_DI_Vars".DI18.xOutput,
           xOutputUnFiltered => "SS2_A3_32DI_DI_Vars".DI18.xInput);
   "DIvars"(xInput := "SS2_A3_32DI_DI_Vars".DI18.xOutput,
            iFuncSystem := "SS2_A3_32DI_DI_Vars".DI18.cFuncSystemID,
            iFuncVar := "SS2_A3_32DI_DI_Vars".DI18.cFuncVar);
END_REGION

REGION Network 19: DIc2 / DI01.1.08 EDP під охороною
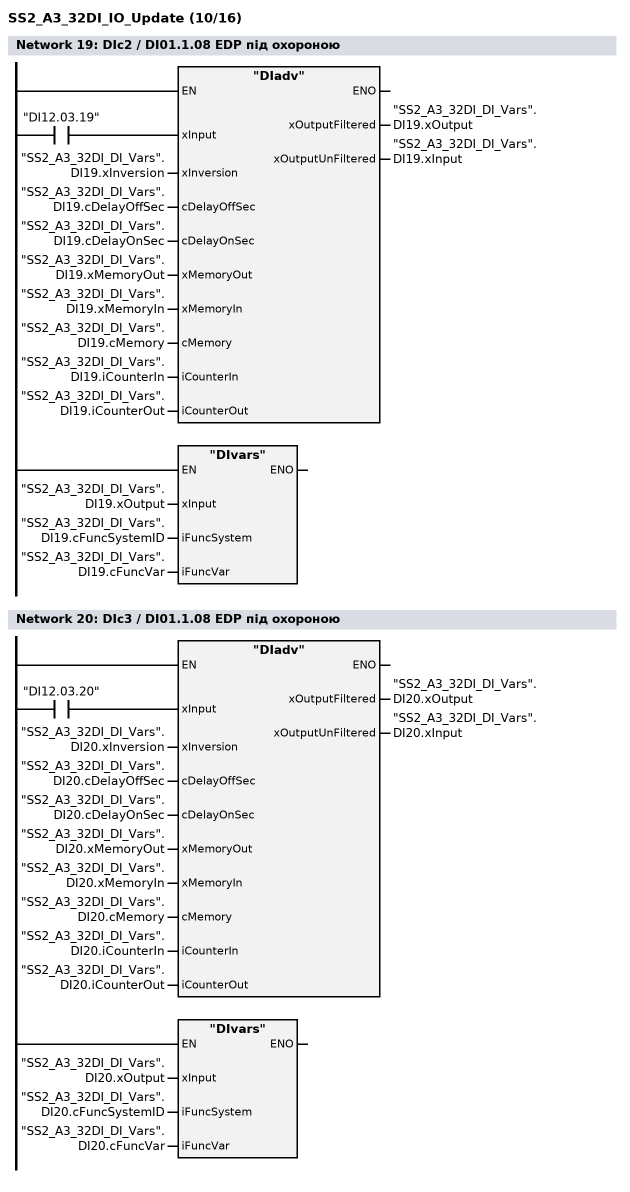
   RUNG wire#powerrail
      "DIadv"(xInput := wire#w1, xInversion := "SS2_A3_32DI_DI_Vars".DI19.xInversion, cDelayOffSec := "SS2_A3_32DI_DI_Vars".DI19.cDelayOffSec, cDelayOnSec := "SS2_A3_32DI_DI_Vars".DI19.cDelayOnSec, xMemoryOut := "SS2_A3_32DI_DI_Vars".DI19.xMemoryOut, xMemoryIn := "SS2_A3_32DI_DI_Vars".DI19.xMemoryIn, cMemory := "SS2_A3_32DI_DI_Vars".DI19.cMemory, iCounterIn := "SS2_A3_32DI_DI_Vars".DI19.iCounterIn, iCounterOut := "SS2_A3_32DI_DI_Vars".DI19.iCounterOut, xOutputFiltered => "SS2_A3_32DI_DI_Vars".DI19.xOutput, xOutputUnFiltered => "SS2_A3_32DI_DI_Vars".DI19.xInput)
   END_RUNG
   RUNG wire#powerrail
      Contact( "DI12.03.19" )
   END_RUNG wire#w1
   RUNG wire#powerrail
      "DIvars"(xInput := "SS2_A3_32DI_DI_Vars".DI19.xOutput, iFuncSystem := "SS2_A3_32DI_DI_Vars".DI19.cFuncSystemID, iFuncVar := "SS2_A3_32DI_DI_Vars".DI19.cFuncVar)
   END_RUNG
   // the same network as SCL:
   "DIadv"(xInput := "DI12.03.19",
           xInversion := "SS2_A3_32DI_DI_Vars".DI19.xInversion,
           cDelayOffSec := "SS2_A3_32DI_DI_Vars".DI19.cDelayOffSec,
           cDelayOnSec := "SS2_A3_32DI_DI_Vars".DI19.cDelayOnSec,
           xMemoryOut := "SS2_A3_32DI_DI_Vars".DI19.xMemoryOut,
           xMemoryIn := "SS2_A3_32DI_DI_Vars".DI19.xMemoryIn,
           cMemory := "SS2_A3_32DI_DI_Vars".DI19.cMemory,
           iCounterIn := "SS2_A3_32DI_DI_Vars".DI19.iCounterIn,
           iCounterOut := "SS2_A3_32DI_DI_Vars".DI19.iCounterOut,
           xOutputFiltered => "SS2_A3_32DI_DI_Vars".DI19.xOutput,
           xOutputUnFiltered => "SS2_A3_32DI_DI_Vars".DI19.xInput);
   "DIvars"(xInput := "SS2_A3_32DI_DI_Vars".DI19.xOutput,
            iFuncSystem := "SS2_A3_32DI_DI_Vars".DI19.cFuncSystemID,
            iFuncVar := "SS2_A3_32DI_DI_Vars".DI19.cFuncVar);
END_REGION

REGION Network 20: DIc3 / DI01.1.08 EDP під охороною
   RUNG wire#powerrail
      "DIadv"(xInput := wire#w1, xInversion := "SS2_A3_32DI_DI_Vars".DI20.xInversion, cDelayOffSec := "SS2_A3_32DI_DI_Vars".DI20.cDelayOffSec, cDelayOnSec := "SS2_A3_32DI_DI_Vars".DI20.cDelayOnSec, xMemoryOut := "SS2_A3_32DI_DI_Vars".DI20.xMemoryOut, xMemoryIn := "SS2_A3_32DI_DI_Vars".DI20.xMemoryIn, cMemory := "SS2_A3_32DI_DI_Vars".DI20.cMemory, iCounterIn := "SS2_A3_32DI_DI_Vars".DI20.iCounterIn, iCounterOut := "SS2_A3_32DI_DI_Vars".DI20.iCounterOut, xOutputFiltered => "SS2_A3_32DI_DI_Vars".DI20.xOutput, xOutputUnFiltered => "SS2_A3_32DI_DI_Vars".DI20.xInput)
   END_RUNG
   RUNG wire#powerrail
      Contact( "DI12.03.20" )
   END_RUNG wire#w1
   RUNG wire#powerrail
      "DIvars"(xInput := "SS2_A3_32DI_DI_Vars".DI20.xOutput, iFuncSystem := "SS2_A3_32DI_DI_Vars".DI20.cFuncSystemID, iFuncVar := "SS2_A3_32DI_DI_Vars".DI20.cFuncVar)
   END_RUNG
   // the same network as SCL:
   "DIadv"(xInput := "DI12.03.20",
           xInversion := "SS2_A3_32DI_DI_Vars".DI20.xInversion,
           cDelayOffSec := "SS2_A3_32DI_DI_Vars".DI20.cDelayOffSec,
           cDelayOnSec := "SS2_A3_32DI_DI_Vars".DI20.cDelayOnSec,
           xMemoryOut := "SS2_A3_32DI_DI_Vars".DI20.xMemoryOut,
           xMemoryIn := "SS2_A3_32DI_DI_Vars".DI20.xMemoryIn,
           cMemory := "SS2_A3_32DI_DI_Vars".DI20.cMemory,
           iCounterIn := "SS2_A3_32DI_DI_Vars".DI20.iCounterIn,
           iCounterOut := "SS2_A3_32DI_DI_Vars".DI20.iCounterOut,
           xOutputFiltered => "SS2_A3_32DI_DI_Vars".DI20.xOutput,
           xOutputUnFiltered => "SS2_A3_32DI_DI_Vars".DI20.xInput);
   "DIvars"(xInput := "SS2_A3_32DI_DI_Vars".DI20.xOutput,
            iFuncSystem := "SS2_A3_32DI_DI_Vars".DI20.cFuncSystemID,
            iFuncVar := "SS2_A3_32DI_DI_Vars".DI20.cFuncVar);
END_REGION

REGION Network 21: DIc4 / DI01.1.08 EDP під охороною
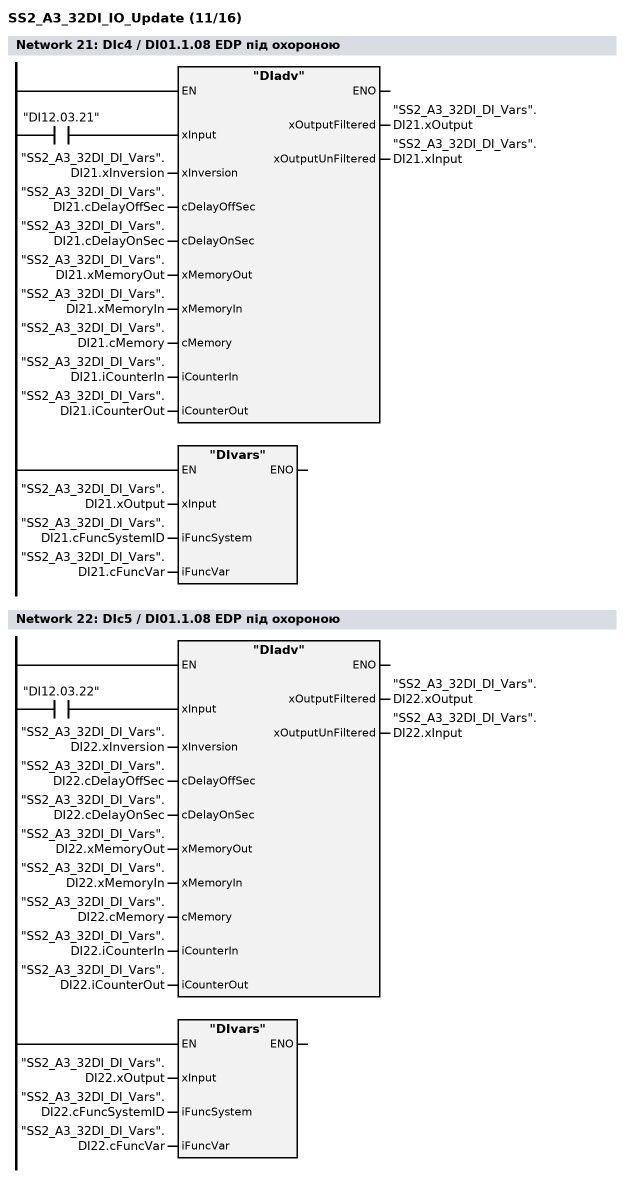
   RUNG wire#powerrail
      "DIadv"(xInput := wire#w1, xInversion := "SS2_A3_32DI_DI_Vars".DI21.xInversion, cDelayOffSec := "SS2_A3_32DI_DI_Vars".DI21.cDelayOffSec, cDelayOnSec := "SS2_A3_32DI_DI_Vars".DI21.cDelayOnSec, xMemoryOut := "SS2_A3_32DI_DI_Vars".DI21.xMemoryOut, xMemoryIn := "SS2_A3_32DI_DI_Vars".DI21.xMemoryIn, cMemory := "SS2_A3_32DI_DI_Vars".DI21.cMemory, iCounterIn := "SS2_A3_32DI_DI_Vars".DI21.iCounterIn, iCounterOut := "SS2_A3_32DI_DI_Vars".DI21.iCounterOut, xOutputFiltered => "SS2_A3_32DI_DI_Vars".DI21.xOutput, xOutputUnFiltered => "SS2_A3_32DI_DI_Vars".DI21.xInput)
   END_RUNG
   RUNG wire#powerrail
      Contact( "DI12.03.21" )
   END_RUNG wire#w1
   RUNG wire#powerrail
      "DIvars"(xInput := "SS2_A3_32DI_DI_Vars".DI21.xOutput, iFuncSystem := "SS2_A3_32DI_DI_Vars".DI21.cFuncSystemID, iFuncVar := "SS2_A3_32DI_DI_Vars".DI21.cFuncVar)
   END_RUNG
   // the same network as SCL:
   "DIadv"(xInput := "DI12.03.21",
           xInversion := "SS2_A3_32DI_DI_Vars".DI21.xInversion,
           cDelayOffSec := "SS2_A3_32DI_DI_Vars".DI21.cDelayOffSec,
           cDelayOnSec := "SS2_A3_32DI_DI_Vars".DI21.cDelayOnSec,
           xMemoryOut := "SS2_A3_32DI_DI_Vars".DI21.xMemoryOut,
           xMemoryIn := "SS2_A3_32DI_DI_Vars".DI21.xMemoryIn,
           cMemory := "SS2_A3_32DI_DI_Vars".DI21.cMemory,
           iCounterIn := "SS2_A3_32DI_DI_Vars".DI21.iCounterIn,
           iCounterOut := "SS2_A3_32DI_DI_Vars".DI21.iCounterOut,
           xOutputFiltered => "SS2_A3_32DI_DI_Vars".DI21.xOutput,
           xOutputUnFiltered => "SS2_A3_32DI_DI_Vars".DI21.xInput);
   "DIvars"(xInput := "SS2_A3_32DI_DI_Vars".DI21.xOutput,
            iFuncSystem := "SS2_A3_32DI_DI_Vars".DI21.cFuncSystemID,
            iFuncVar := "SS2_A3_32DI_DI_Vars".DI21.cFuncVar);
END_REGION

REGION Network 22: DIc5 / DI01.1.08 EDP під охороною
   RUNG wire#powerrail
      "DIadv"(xInput := wire#w1, xInversion := "SS2_A3_32DI_DI_Vars".DI22.xInversion, cDelayOffSec := "SS2_A3_32DI_DI_Vars".DI22.cDelayOffSec, cDelayOnSec := "SS2_A3_32DI_DI_Vars".DI22.cDelayOnSec, xMemoryOut := "SS2_A3_32DI_DI_Vars".DI22.xMemoryOut, xMemoryIn := "SS2_A3_32DI_DI_Vars".DI22.xMemoryIn, cMemory := "SS2_A3_32DI_DI_Vars".DI22.cMemory, iCounterIn := "SS2_A3_32DI_DI_Vars".DI22.iCounterIn, iCounterOut := "SS2_A3_32DI_DI_Vars".DI22.iCounterOut, xOutputFiltered => "SS2_A3_32DI_DI_Vars".DI22.xOutput, xOutputUnFiltered => "SS2_A3_32DI_DI_Vars".DI22.xInput)
   END_RUNG
   RUNG wire#powerrail
      Contact( "DI12.03.22" )
   END_RUNG wire#w1
   RUNG wire#powerrail
      "DIvars"(xInput := "SS2_A3_32DI_DI_Vars".DI22.xOutput, iFuncSystem := "SS2_A3_32DI_DI_Vars".DI22.cFuncSystemID, iFuncVar := "SS2_A3_32DI_DI_Vars".DI22.cFuncVar)
   END_RUNG
   // the same network as SCL:
   "DIadv"(xInput := "DI12.03.22",
           xInversion := "SS2_A3_32DI_DI_Vars".DI22.xInversion,
           cDelayOffSec := "SS2_A3_32DI_DI_Vars".DI22.cDelayOffSec,
           cDelayOnSec := "SS2_A3_32DI_DI_Vars".DI22.cDelayOnSec,
           xMemoryOut := "SS2_A3_32DI_DI_Vars".DI22.xMemoryOut,
           xMemoryIn := "SS2_A3_32DI_DI_Vars".DI22.xMemoryIn,
           cMemory := "SS2_A3_32DI_DI_Vars".DI22.cMemory,
           iCounterIn := "SS2_A3_32DI_DI_Vars".DI22.iCounterIn,
           iCounterOut := "SS2_A3_32DI_DI_Vars".DI22.iCounterOut,
           xOutputFiltered => "SS2_A3_32DI_DI_Vars".DI22.xOutput,
           xOutputUnFiltered => "SS2_A3_32DI_DI_Vars".DI22.xInput);
   "DIvars"(xInput := "SS2_A3_32DI_DI_Vars".DI22.xOutput,
            iFuncSystem := "SS2_A3_32DI_DI_Vars".DI22.cFuncSystemID,
            iFuncVar := "SS2_A3_32DI_DI_Vars".DI22.cFuncVar);
END_REGION

REGION Network 23: DIc6 / DI01.1.08 EDP під охороною
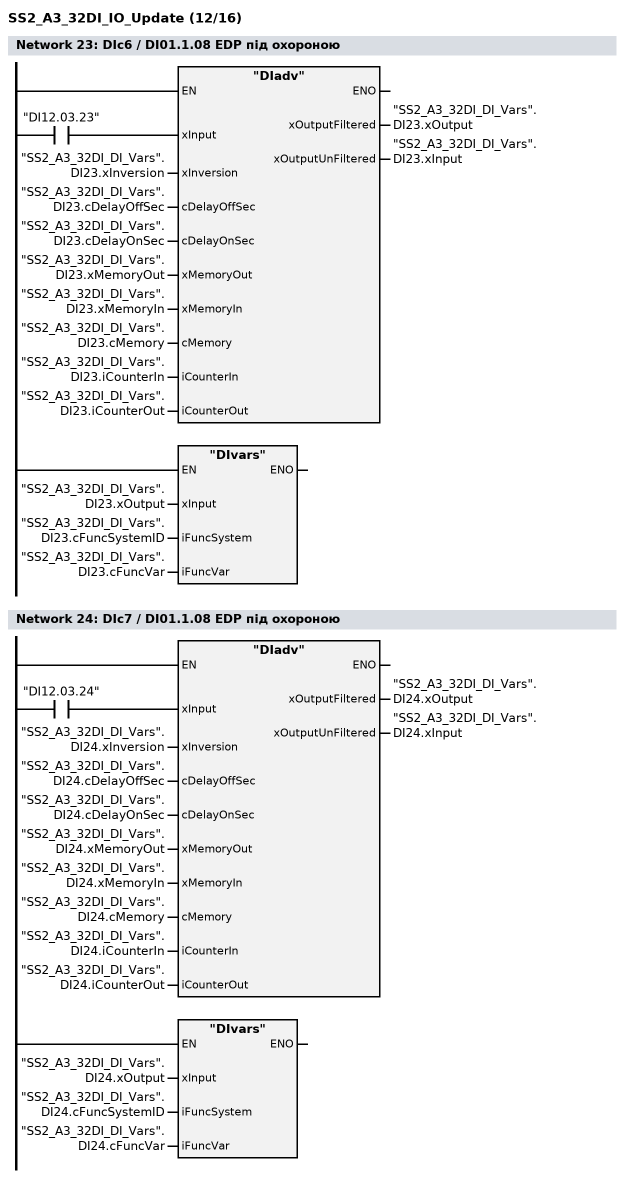
   RUNG wire#powerrail
      "DIadv"(xInput := wire#w1, xInversion := "SS2_A3_32DI_DI_Vars".DI23.xInversion, cDelayOffSec := "SS2_A3_32DI_DI_Vars".DI23.cDelayOffSec, cDelayOnSec := "SS2_A3_32DI_DI_Vars".DI23.cDelayOnSec, xMemoryOut := "SS2_A3_32DI_DI_Vars".DI23.xMemoryOut, xMemoryIn := "SS2_A3_32DI_DI_Vars".DI23.xMemoryIn, cMemory := "SS2_A3_32DI_DI_Vars".DI23.cMemory, iCounterIn := "SS2_A3_32DI_DI_Vars".DI23.iCounterIn, iCounterOut := "SS2_A3_32DI_DI_Vars".DI23.iCounterOut, xOutputFiltered => "SS2_A3_32DI_DI_Vars".DI23.xOutput, xOutputUnFiltered => "SS2_A3_32DI_DI_Vars".DI23.xInput)
   END_RUNG
   RUNG wire#powerrail
      Contact( "DI12.03.23" )
   END_RUNG wire#w1
   RUNG wire#powerrail
      "DIvars"(xInput := "SS2_A3_32DI_DI_Vars".DI23.xOutput, iFuncSystem := "SS2_A3_32DI_DI_Vars".DI23.cFuncSystemID, iFuncVar := "SS2_A3_32DI_DI_Vars".DI23.cFuncVar)
   END_RUNG
   // the same network as SCL:
   "DIadv"(xInput := "DI12.03.23",
           xInversion := "SS2_A3_32DI_DI_Vars".DI23.xInversion,
           cDelayOffSec := "SS2_A3_32DI_DI_Vars".DI23.cDelayOffSec,
           cDelayOnSec := "SS2_A3_32DI_DI_Vars".DI23.cDelayOnSec,
           xMemoryOut := "SS2_A3_32DI_DI_Vars".DI23.xMemoryOut,
           xMemoryIn := "SS2_A3_32DI_DI_Vars".DI23.xMemoryIn,
           cMemory := "SS2_A3_32DI_DI_Vars".DI23.cMemory,
           iCounterIn := "SS2_A3_32DI_DI_Vars".DI23.iCounterIn,
           iCounterOut := "SS2_A3_32DI_DI_Vars".DI23.iCounterOut,
           xOutputFiltered => "SS2_A3_32DI_DI_Vars".DI23.xOutput,
           xOutputUnFiltered => "SS2_A3_32DI_DI_Vars".DI23.xInput);
   "DIvars"(xInput := "SS2_A3_32DI_DI_Vars".DI23.xOutput,
            iFuncSystem := "SS2_A3_32DI_DI_Vars".DI23.cFuncSystemID,
            iFuncVar := "SS2_A3_32DI_DI_Vars".DI23.cFuncVar);
END_REGION

REGION Network 24: DIc7 / DI01.1.08 EDP під охороною
   RUNG wire#powerrail
      "DIadv"(xInput := wire#w1, xInversion := "SS2_A3_32DI_DI_Vars".DI24.xInversion, cDelayOffSec := "SS2_A3_32DI_DI_Vars".DI24.cDelayOffSec, cDelayOnSec := "SS2_A3_32DI_DI_Vars".DI24.cDelayOnSec, xMemoryOut := "SS2_A3_32DI_DI_Vars".DI24.xMemoryOut, xMemoryIn := "SS2_A3_32DI_DI_Vars".DI24.xMemoryIn, cMemory := "SS2_A3_32DI_DI_Vars".DI24.cMemory, iCounterIn := "SS2_A3_32DI_DI_Vars".DI24.iCounterIn, iCounterOut := "SS2_A3_32DI_DI_Vars".DI24.iCounterOut, xOutputFiltered => "SS2_A3_32DI_DI_Vars".DI24.xOutput, xOutputUnFiltered => "SS2_A3_32DI_DI_Vars".DI24.xInput)
   END_RUNG
   RUNG wire#powerrail
      Contact( "DI12.03.24" )
   END_RUNG wire#w1
   RUNG wire#powerrail
      "DIvars"(xInput := "SS2_A3_32DI_DI_Vars".DI24.xOutput, iFuncSystem := "SS2_A3_32DI_DI_Vars".DI24.cFuncSystemID, iFuncVar := "SS2_A3_32DI_DI_Vars".DI24.cFuncVar)
   END_RUNG
   // the same network as SCL:
   "DIadv"(xInput := "DI12.03.24",
           xInversion := "SS2_A3_32DI_DI_Vars".DI24.xInversion,
           cDelayOffSec := "SS2_A3_32DI_DI_Vars".DI24.cDelayOffSec,
           cDelayOnSec := "SS2_A3_32DI_DI_Vars".DI24.cDelayOnSec,
           xMemoryOut := "SS2_A3_32DI_DI_Vars".DI24.xMemoryOut,
           xMemoryIn := "SS2_A3_32DI_DI_Vars".DI24.xMemoryIn,
           cMemory := "SS2_A3_32DI_DI_Vars".DI24.cMemory,
           iCounterIn := "SS2_A3_32DI_DI_Vars".DI24.iCounterIn,
           iCounterOut := "SS2_A3_32DI_DI_Vars".DI24.iCounterOut,
           xOutputFiltered => "SS2_A3_32DI_DI_Vars".DI24.xOutput,
           xOutputUnFiltered => "SS2_A3_32DI_DI_Vars".DI24.xInput);
   "DIvars"(xInput := "SS2_A3_32DI_DI_Vars".DI24.xOutput,
            iFuncSystem := "SS2_A3_32DI_DI_Vars".DI24.cFuncSystemID,
            iFuncVar := "SS2_A3_32DI_DI_Vars".DI24.cFuncVar);
END_REGION

REGION Network 25: DId0 / DI01.1.08 EDP під охороною
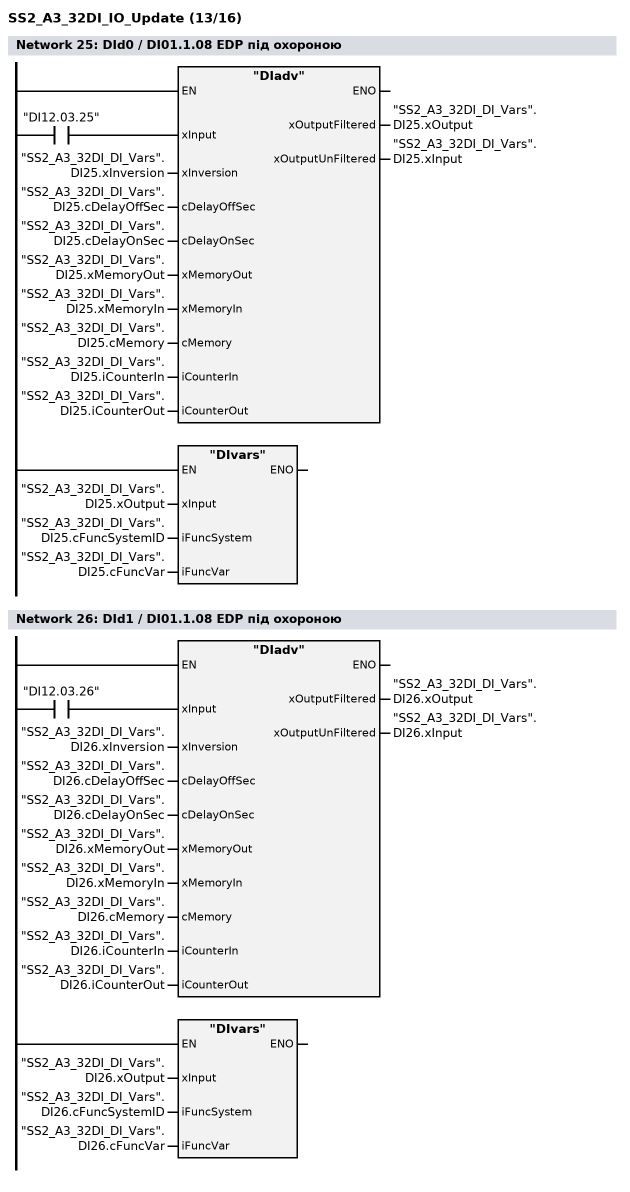
   RUNG wire#powerrail
      "DIadv"(xInput := wire#w1, xInversion := "SS2_A3_32DI_DI_Vars".DI25.xInversion, cDelayOffSec := "SS2_A3_32DI_DI_Vars".DI25.cDelayOffSec, cDelayOnSec := "SS2_A3_32DI_DI_Vars".DI25.cDelayOnSec, xMemoryOut := "SS2_A3_32DI_DI_Vars".DI25.xMemoryOut, xMemoryIn := "SS2_A3_32DI_DI_Vars".DI25.xMemoryIn, cMemory := "SS2_A3_32DI_DI_Vars".DI25.cMemory, iCounterIn := "SS2_A3_32DI_DI_Vars".DI25.iCounterIn, iCounterOut := "SS2_A3_32DI_DI_Vars".DI25.iCounterOut, xOutputFiltered => "SS2_A3_32DI_DI_Vars".DI25.xOutput, xOutputUnFiltered => "SS2_A3_32DI_DI_Vars".DI25.xInput)
   END_RUNG
   RUNG wire#powerrail
      Contact( "DI12.03.25" )
   END_RUNG wire#w1
   RUNG wire#powerrail
      "DIvars"(xInput := "SS2_A3_32DI_DI_Vars".DI25.xOutput, iFuncSystem := "SS2_A3_32DI_DI_Vars".DI25.cFuncSystemID, iFuncVar := "SS2_A3_32DI_DI_Vars".DI25.cFuncVar)
   END_RUNG
   // the same network as SCL:
   "DIadv"(xInput := "DI12.03.25",
           xInversion := "SS2_A3_32DI_DI_Vars".DI25.xInversion,
           cDelayOffSec := "SS2_A3_32DI_DI_Vars".DI25.cDelayOffSec,
           cDelayOnSec := "SS2_A3_32DI_DI_Vars".DI25.cDelayOnSec,
           xMemoryOut := "SS2_A3_32DI_DI_Vars".DI25.xMemoryOut,
           xMemoryIn := "SS2_A3_32DI_DI_Vars".DI25.xMemoryIn,
           cMemory := "SS2_A3_32DI_DI_Vars".DI25.cMemory,
           iCounterIn := "SS2_A3_32DI_DI_Vars".DI25.iCounterIn,
           iCounterOut := "SS2_A3_32DI_DI_Vars".DI25.iCounterOut,
           xOutputFiltered => "SS2_A3_32DI_DI_Vars".DI25.xOutput,
           xOutputUnFiltered => "SS2_A3_32DI_DI_Vars".DI25.xInput);
   "DIvars"(xInput := "SS2_A3_32DI_DI_Vars".DI25.xOutput,
            iFuncSystem := "SS2_A3_32DI_DI_Vars".DI25.cFuncSystemID,
            iFuncVar := "SS2_A3_32DI_DI_Vars".DI25.cFuncVar);
END_REGION

REGION Network 26: DId1 / DI01.1.08 EDP під охороною
   RUNG wire#powerrail
      "DIadv"(xInput := wire#w1, xInversion := "SS2_A3_32DI_DI_Vars".DI26.xInversion, cDelayOffSec := "SS2_A3_32DI_DI_Vars".DI26.cDelayOffSec, cDelayOnSec := "SS2_A3_32DI_DI_Vars".DI26.cDelayOnSec, xMemoryOut := "SS2_A3_32DI_DI_Vars".DI26.xMemoryOut, xMemoryIn := "SS2_A3_32DI_DI_Vars".DI26.xMemoryIn, cMemory := "SS2_A3_32DI_DI_Vars".DI26.cMemory, iCounterIn := "SS2_A3_32DI_DI_Vars".DI26.iCounterIn, iCounterOut := "SS2_A3_32DI_DI_Vars".DI26.iCounterOut, xOutputFiltered => "SS2_A3_32DI_DI_Vars".DI26.xOutput, xOutputUnFiltered => "SS2_A3_32DI_DI_Vars".DI26.xInput)
   END_RUNG
   RUNG wire#powerrail
      Contact( "DI12.03.26" )
   END_RUNG wire#w1
   RUNG wire#powerrail
      "DIvars"(xInput := "SS2_A3_32DI_DI_Vars".DI26.xOutput, iFuncSystem := "SS2_A3_32DI_DI_Vars".DI26.cFuncSystemID, iFuncVar := "SS2_A3_32DI_DI_Vars".DI26.cFuncVar)
   END_RUNG
   // the same network as SCL:
   "DIadv"(xInput := "DI12.03.26",
           xInversion := "SS2_A3_32DI_DI_Vars".DI26.xInversion,
           cDelayOffSec := "SS2_A3_32DI_DI_Vars".DI26.cDelayOffSec,
           cDelayOnSec := "SS2_A3_32DI_DI_Vars".DI26.cDelayOnSec,
           xMemoryOut := "SS2_A3_32DI_DI_Vars".DI26.xMemoryOut,
           xMemoryIn := "SS2_A3_32DI_DI_Vars".DI26.xMemoryIn,
           cMemory := "SS2_A3_32DI_DI_Vars".DI26.cMemory,
           iCounterIn := "SS2_A3_32DI_DI_Vars".DI26.iCounterIn,
           iCounterOut := "SS2_A3_32DI_DI_Vars".DI26.iCounterOut,
           xOutputFiltered => "SS2_A3_32DI_DI_Vars".DI26.xOutput,
           xOutputUnFiltered => "SS2_A3_32DI_DI_Vars".DI26.xInput);
   "DIvars"(xInput := "SS2_A3_32DI_DI_Vars".DI26.xOutput,
            iFuncSystem := "SS2_A3_32DI_DI_Vars".DI26.cFuncSystemID,
            iFuncVar := "SS2_A3_32DI_DI_Vars".DI26.cFuncVar);
END_REGION

REGION Network 27: DId2 / DI01.1.08 EDP під охороною
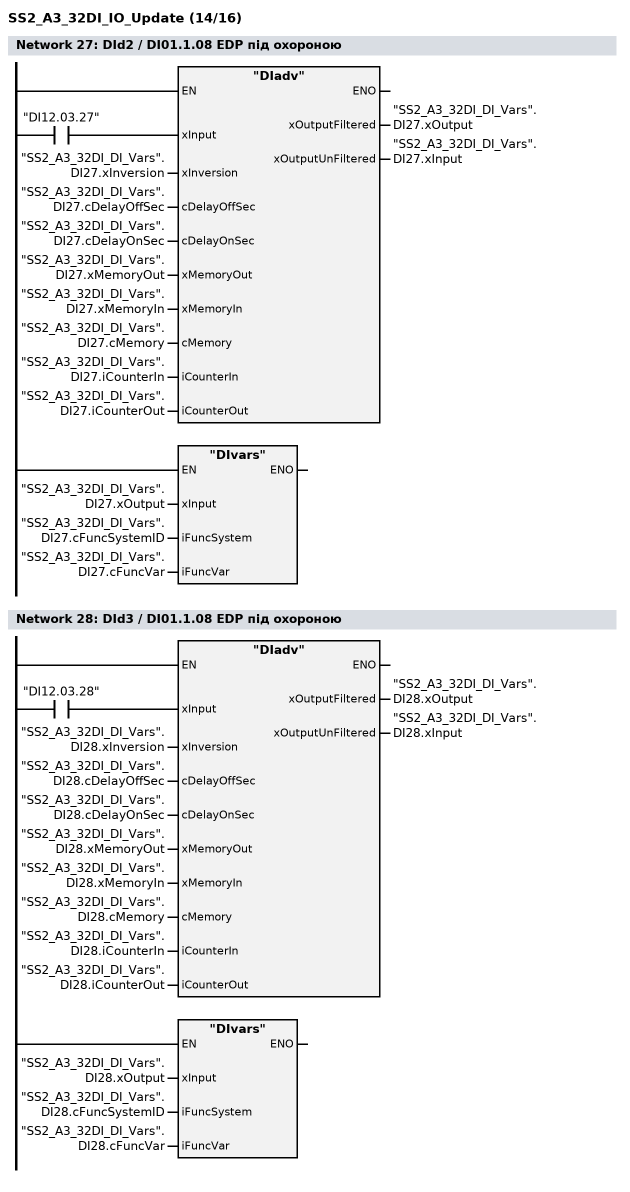
   RUNG wire#powerrail
      "DIadv"(xInput := wire#w1, xInversion := "SS2_A3_32DI_DI_Vars".DI27.xInversion, cDelayOffSec := "SS2_A3_32DI_DI_Vars".DI27.cDelayOffSec, cDelayOnSec := "SS2_A3_32DI_DI_Vars".DI27.cDelayOnSec, xMemoryOut := "SS2_A3_32DI_DI_Vars".DI27.xMemoryOut, xMemoryIn := "SS2_A3_32DI_DI_Vars".DI27.xMemoryIn, cMemory := "SS2_A3_32DI_DI_Vars".DI27.cMemory, iCounterIn := "SS2_A3_32DI_DI_Vars".DI27.iCounterIn, iCounterOut := "SS2_A3_32DI_DI_Vars".DI27.iCounterOut, xOutputFiltered => "SS2_A3_32DI_DI_Vars".DI27.xOutput, xOutputUnFiltered => "SS2_A3_32DI_DI_Vars".DI27.xInput)
   END_RUNG
   RUNG wire#powerrail
      Contact( "DI12.03.27" )
   END_RUNG wire#w1
   RUNG wire#powerrail
      "DIvars"(xInput := "SS2_A3_32DI_DI_Vars".DI27.xOutput, iFuncSystem := "SS2_A3_32DI_DI_Vars".DI27.cFuncSystemID, iFuncVar := "SS2_A3_32DI_DI_Vars".DI27.cFuncVar)
   END_RUNG
   // the same network as SCL:
   "DIadv"(xInput := "DI12.03.27",
           xInversion := "SS2_A3_32DI_DI_Vars".DI27.xInversion,
           cDelayOffSec := "SS2_A3_32DI_DI_Vars".DI27.cDelayOffSec,
           cDelayOnSec := "SS2_A3_32DI_DI_Vars".DI27.cDelayOnSec,
           xMemoryOut := "SS2_A3_32DI_DI_Vars".DI27.xMemoryOut,
           xMemoryIn := "SS2_A3_32DI_DI_Vars".DI27.xMemoryIn,
           cMemory := "SS2_A3_32DI_DI_Vars".DI27.cMemory,
           iCounterIn := "SS2_A3_32DI_DI_Vars".DI27.iCounterIn,
           iCounterOut := "SS2_A3_32DI_DI_Vars".DI27.iCounterOut,
           xOutputFiltered => "SS2_A3_32DI_DI_Vars".DI27.xOutput,
           xOutputUnFiltered => "SS2_A3_32DI_DI_Vars".DI27.xInput);
   "DIvars"(xInput := "SS2_A3_32DI_DI_Vars".DI27.xOutput,
            iFuncSystem := "SS2_A3_32DI_DI_Vars".DI27.cFuncSystemID,
            iFuncVar := "SS2_A3_32DI_DI_Vars".DI27.cFuncVar);
END_REGION

REGION Network 28: DId3 / DI01.1.08 EDP під охороною
   RUNG wire#powerrail
      "DIadv"(xInput := wire#w1, xInversion := "SS2_A3_32DI_DI_Vars".DI28.xInversion, cDelayOffSec := "SS2_A3_32DI_DI_Vars".DI28.cDelayOffSec, cDelayOnSec := "SS2_A3_32DI_DI_Vars".DI28.cDelayOnSec, xMemoryOut := "SS2_A3_32DI_DI_Vars".DI28.xMemoryOut, xMemoryIn := "SS2_A3_32DI_DI_Vars".DI28.xMemoryIn, cMemory := "SS2_A3_32DI_DI_Vars".DI28.cMemory, iCounterIn := "SS2_A3_32DI_DI_Vars".DI28.iCounterIn, iCounterOut := "SS2_A3_32DI_DI_Vars".DI28.iCounterOut, xOutputFiltered => "SS2_A3_32DI_DI_Vars".DI28.xOutput, xOutputUnFiltered => "SS2_A3_32DI_DI_Vars".DI28.xInput)
   END_RUNG
   RUNG wire#powerrail
      Contact( "DI12.03.28" )
   END_RUNG wire#w1
   RUNG wire#powerrail
      "DIvars"(xInput := "SS2_A3_32DI_DI_Vars".DI28.xOutput, iFuncSystem := "SS2_A3_32DI_DI_Vars".DI28.cFuncSystemID, iFuncVar := "SS2_A3_32DI_DI_Vars".DI28.cFuncVar)
   END_RUNG
   // the same network as SCL:
   "DIadv"(xInput := "DI12.03.28",
           xInversion := "SS2_A3_32DI_DI_Vars".DI28.xInversion,
           cDelayOffSec := "SS2_A3_32DI_DI_Vars".DI28.cDelayOffSec,
           cDelayOnSec := "SS2_A3_32DI_DI_Vars".DI28.cDelayOnSec,
           xMemoryOut := "SS2_A3_32DI_DI_Vars".DI28.xMemoryOut,
           xMemoryIn := "SS2_A3_32DI_DI_Vars".DI28.xMemoryIn,
           cMemory := "SS2_A3_32DI_DI_Vars".DI28.cMemory,
           iCounterIn := "SS2_A3_32DI_DI_Vars".DI28.iCounterIn,
           iCounterOut := "SS2_A3_32DI_DI_Vars".DI28.iCounterOut,
           xOutputFiltered => "SS2_A3_32DI_DI_Vars".DI28.xOutput,
           xOutputUnFiltered => "SS2_A3_32DI_DI_Vars".DI28.xInput);
   "DIvars"(xInput := "SS2_A3_32DI_DI_Vars".DI28.xOutput,
            iFuncSystem := "SS2_A3_32DI_DI_Vars".DI28.cFuncSystemID,
            iFuncVar := "SS2_A3_32DI_DI_Vars".DI28.cFuncVar);
END_REGION

REGION Network 29: DId4 / DI01.1.08 EDP під охороною
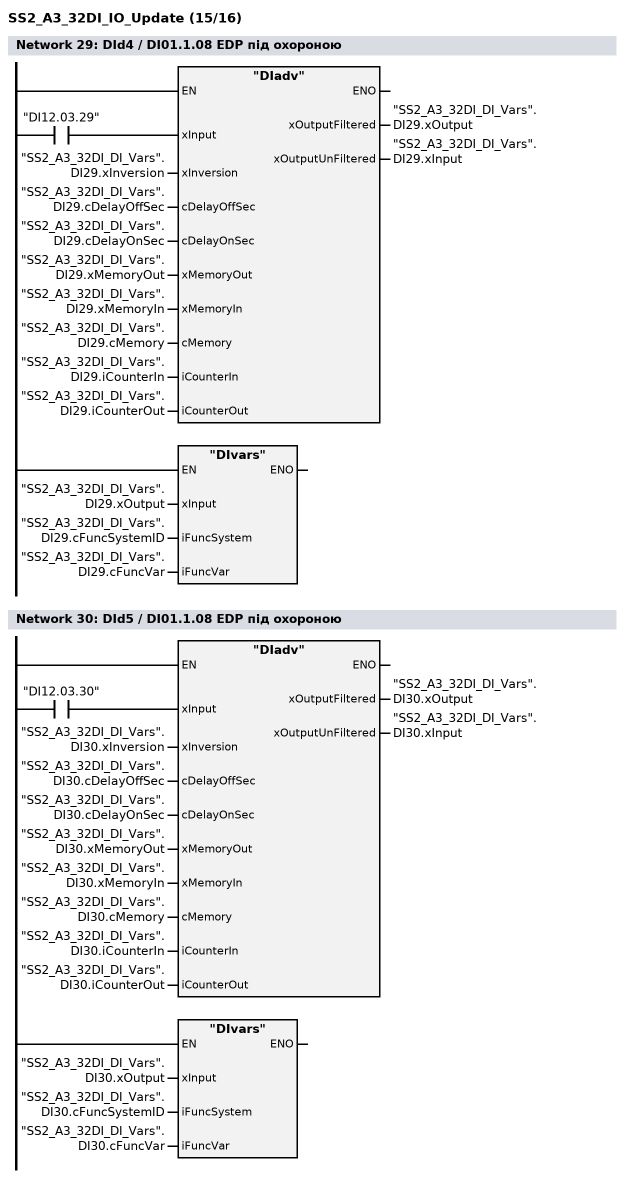
   RUNG wire#powerrail
      "DIadv"(xInput := wire#w1, xInversion := "SS2_A3_32DI_DI_Vars".DI29.xInversion, cDelayOffSec := "SS2_A3_32DI_DI_Vars".DI29.cDelayOffSec, cDelayOnSec := "SS2_A3_32DI_DI_Vars".DI29.cDelayOnSec, xMemoryOut := "SS2_A3_32DI_DI_Vars".DI29.xMemoryOut, xMemoryIn := "SS2_A3_32DI_DI_Vars".DI29.xMemoryIn, cMemory := "SS2_A3_32DI_DI_Vars".DI29.cMemory, iCounterIn := "SS2_A3_32DI_DI_Vars".DI29.iCounterIn, iCounterOut := "SS2_A3_32DI_DI_Vars".DI29.iCounterOut, xOutputFiltered => "SS2_A3_32DI_DI_Vars".DI29.xOutput, xOutputUnFiltered => "SS2_A3_32DI_DI_Vars".DI29.xInput)
   END_RUNG
   RUNG wire#powerrail
      Contact( "DI12.03.29" )
   END_RUNG wire#w1
   RUNG wire#powerrail
      "DIvars"(xInput := "SS2_A3_32DI_DI_Vars".DI29.xOutput, iFuncSystem := "SS2_A3_32DI_DI_Vars".DI29.cFuncSystemID, iFuncVar := "SS2_A3_32DI_DI_Vars".DI29.cFuncVar)
   END_RUNG
   // the same network as SCL:
   "DIadv"(xInput := "DI12.03.29",
           xInversion := "SS2_A3_32DI_DI_Vars".DI29.xInversion,
           cDelayOffSec := "SS2_A3_32DI_DI_Vars".DI29.cDelayOffSec,
           cDelayOnSec := "SS2_A3_32DI_DI_Vars".DI29.cDelayOnSec,
           xMemoryOut := "SS2_A3_32DI_DI_Vars".DI29.xMemoryOut,
           xMemoryIn := "SS2_A3_32DI_DI_Vars".DI29.xMemoryIn,
           cMemory := "SS2_A3_32DI_DI_Vars".DI29.cMemory,
           iCounterIn := "SS2_A3_32DI_DI_Vars".DI29.iCounterIn,
           iCounterOut := "SS2_A3_32DI_DI_Vars".DI29.iCounterOut,
           xOutputFiltered => "SS2_A3_32DI_DI_Vars".DI29.xOutput,
           xOutputUnFiltered => "SS2_A3_32DI_DI_Vars".DI29.xInput);
   "DIvars"(xInput := "SS2_A3_32DI_DI_Vars".DI29.xOutput,
            iFuncSystem := "SS2_A3_32DI_DI_Vars".DI29.cFuncSystemID,
            iFuncVar := "SS2_A3_32DI_DI_Vars".DI29.cFuncVar);
END_REGION

REGION Network 30: DId5 / DI01.1.08 EDP під охороною
   RUNG wire#powerrail
      "DIadv"(xInput := wire#w1, xInversion := "SS2_A3_32DI_DI_Vars".DI30.xInversion, cDelayOffSec := "SS2_A3_32DI_DI_Vars".DI30.cDelayOffSec, cDelayOnSec := "SS2_A3_32DI_DI_Vars".DI30.cDelayOnSec, xMemoryOut := "SS2_A3_32DI_DI_Vars".DI30.xMemoryOut, xMemoryIn := "SS2_A3_32DI_DI_Vars".DI30.xMemoryIn, cMemory := "SS2_A3_32DI_DI_Vars".DI30.cMemory, iCounterIn := "SS2_A3_32DI_DI_Vars".DI30.iCounterIn, iCounterOut := "SS2_A3_32DI_DI_Vars".DI30.iCounterOut, xOutputFiltered => "SS2_A3_32DI_DI_Vars".DI30.xOutput, xOutputUnFiltered => "SS2_A3_32DI_DI_Vars".DI30.xInput)
   END_RUNG
   RUNG wire#powerrail
      Contact( "DI12.03.30" )
   END_RUNG wire#w1
   RUNG wire#powerrail
      "DIvars"(xInput := "SS2_A3_32DI_DI_Vars".DI30.xOutput, iFuncSystem := "SS2_A3_32DI_DI_Vars".DI30.cFuncSystemID, iFuncVar := "SS2_A3_32DI_DI_Vars".DI30.cFuncVar)
   END_RUNG
   // the same network as SCL:
   "DIadv"(xInput := "DI12.03.30",
           xInversion := "SS2_A3_32DI_DI_Vars".DI30.xInversion,
           cDelayOffSec := "SS2_A3_32DI_DI_Vars".DI30.cDelayOffSec,
           cDelayOnSec := "SS2_A3_32DI_DI_Vars".DI30.cDelayOnSec,
           xMemoryOut := "SS2_A3_32DI_DI_Vars".DI30.xMemoryOut,
           xMemoryIn := "SS2_A3_32DI_DI_Vars".DI30.xMemoryIn,
           cMemory := "SS2_A3_32DI_DI_Vars".DI30.cMemory,
           iCounterIn := "SS2_A3_32DI_DI_Vars".DI30.iCounterIn,
           iCounterOut := "SS2_A3_32DI_DI_Vars".DI30.iCounterOut,
           xOutputFiltered => "SS2_A3_32DI_DI_Vars".DI30.xOutput,
           xOutputUnFiltered => "SS2_A3_32DI_DI_Vars".DI30.xInput);
   "DIvars"(xInput := "SS2_A3_32DI_DI_Vars".DI30.xOutput,
            iFuncSystem := "SS2_A3_32DI_DI_Vars".DI30.cFuncSystemID,
            iFuncVar := "SS2_A3_32DI_DI_Vars".DI30.cFuncVar);
END_REGION

REGION Network 31: DId6 / DI01.1.08 EDP під охороною
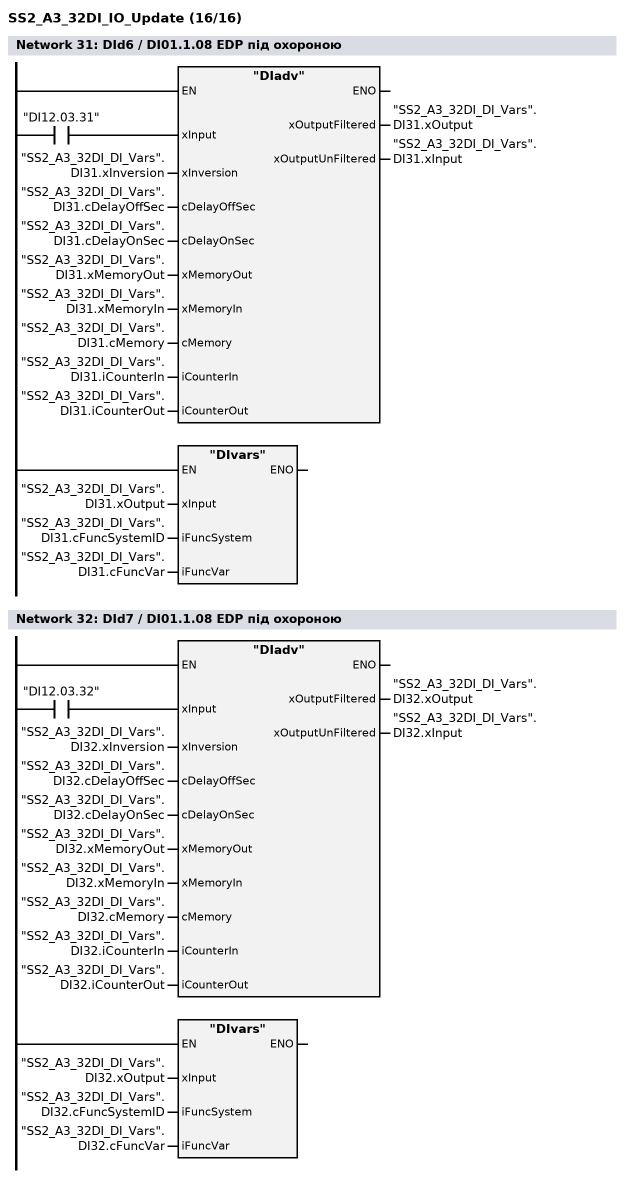
   RUNG wire#powerrail
      "DIadv"(xInput := wire#w1, xInversion := "SS2_A3_32DI_DI_Vars".DI31.xInversion, cDelayOffSec := "SS2_A3_32DI_DI_Vars".DI31.cDelayOffSec, cDelayOnSec := "SS2_A3_32DI_DI_Vars".DI31.cDelayOnSec, xMemoryOut := "SS2_A3_32DI_DI_Vars".DI31.xMemoryOut, xMemoryIn := "SS2_A3_32DI_DI_Vars".DI31.xMemoryIn, cMemory := "SS2_A3_32DI_DI_Vars".DI31.cMemory, iCounterIn := "SS2_A3_32DI_DI_Vars".DI31.iCounterIn, iCounterOut := "SS2_A3_32DI_DI_Vars".DI31.iCounterOut, xOutputFiltered => "SS2_A3_32DI_DI_Vars".DI31.xOutput, xOutputUnFiltered => "SS2_A3_32DI_DI_Vars".DI31.xInput)
   END_RUNG
   RUNG wire#powerrail
      Contact( "DI12.03.31" )
   END_RUNG wire#w1
   RUNG wire#powerrail
      "DIvars"(xInput := "SS2_A3_32DI_DI_Vars".DI31.xOutput, iFuncSystem := "SS2_A3_32DI_DI_Vars".DI31.cFuncSystemID, iFuncVar := "SS2_A3_32DI_DI_Vars".DI31.cFuncVar)
   END_RUNG
   // the same network as SCL:
   "DIadv"(xInput := "DI12.03.31",
           xInversion := "SS2_A3_32DI_DI_Vars".DI31.xInversion,
           cDelayOffSec := "SS2_A3_32DI_DI_Vars".DI31.cDelayOffSec,
           cDelayOnSec := "SS2_A3_32DI_DI_Vars".DI31.cDelayOnSec,
           xMemoryOut := "SS2_A3_32DI_DI_Vars".DI31.xMemoryOut,
           xMemoryIn := "SS2_A3_32DI_DI_Vars".DI31.xMemoryIn,
           cMemory := "SS2_A3_32DI_DI_Vars".DI31.cMemory,
           iCounterIn := "SS2_A3_32DI_DI_Vars".DI31.iCounterIn,
           iCounterOut := "SS2_A3_32DI_DI_Vars".DI31.iCounterOut,
           xOutputFiltered => "SS2_A3_32DI_DI_Vars".DI31.xOutput,
           xOutputUnFiltered => "SS2_A3_32DI_DI_Vars".DI31.xInput);
   "DIvars"(xInput := "SS2_A3_32DI_DI_Vars".DI31.xOutput,
            iFuncSystem := "SS2_A3_32DI_DI_Vars".DI31.cFuncSystemID,
            iFuncVar := "SS2_A3_32DI_DI_Vars".DI31.cFuncVar);
END_REGION

REGION Network 32: DId7 / DI01.1.08 EDP під охороною
   RUNG wire#powerrail
      "DIadv"(xInput := wire#w1, xInversion := "SS2_A3_32DI_DI_Vars".DI32.xInversion, cDelayOffSec := "SS2_A3_32DI_DI_Vars".DI32.cDelayOffSec, cDelayOnSec := "SS2_A3_32DI_DI_Vars".DI32.cDelayOnSec, xMemoryOut := "SS2_A3_32DI_DI_Vars".DI32.xMemoryOut, xMemoryIn := "SS2_A3_32DI_DI_Vars".DI32.xMemoryIn, cMemory := "SS2_A3_32DI_DI_Vars".DI32.cMemory, iCounterIn := "SS2_A3_32DI_DI_Vars".DI32.iCounterIn, iCounterOut := "SS2_A3_32DI_DI_Vars".DI32.iCounterOut, xOutputFiltered => "SS2_A3_32DI_DI_Vars".DI32.xOutput, xOutputUnFiltered => "SS2_A3_32DI_DI_Vars".DI32.xInput)
   END_RUNG
   RUNG wire#powerrail
      Contact( "DI12.03.32" )
   END_RUNG wire#w1
   RUNG wire#powerrail
      "DIvars"(xInput := "SS2_A3_32DI_DI_Vars".DI32.xOutput, iFuncSystem := "SS2_A3_32DI_DI_Vars".DI32.cFuncSystemID, iFuncVar := "SS2_A3_32DI_DI_Vars".DI32.cFuncVar)
   END_RUNG
   // the same network as SCL:
   "DIadv"(xInput := "DI12.03.32",
           xInversion := "SS2_A3_32DI_DI_Vars".DI32.xInversion,
           cDelayOffSec := "SS2_A3_32DI_DI_Vars".DI32.cDelayOffSec,
           cDelayOnSec := "SS2_A3_32DI_DI_Vars".DI32.cDelayOnSec,
           xMemoryOut := "SS2_A3_32DI_DI_Vars".DI32.xMemoryOut,
           xMemoryIn := "SS2_A3_32DI_DI_Vars".DI32.xMemoryIn,
           cMemory := "SS2_A3_32DI_DI_Vars".DI32.cMemory,
           iCounterIn := "SS2_A3_32DI_DI_Vars".DI32.iCounterIn,
           iCounterOut := "SS2_A3_32DI_DI_Vars".DI32.iCounterOut,
           xOutputFiltered => "SS2_A3_32DI_DI_Vars".DI32.xOutput,
           xOutputUnFiltered => "SS2_A3_32DI_DI_Vars".DI32.xInput);
   "DIvars"(xInput := "SS2_A3_32DI_DI_Vars".DI32.xOutput,
            iFuncSystem := "SS2_A3_32DI_DI_Vars".DI32.cFuncSystemID,
            iFuncVar := "SS2_A3_32DI_DI_Vars".DI32.cFuncVar);
END_REGION
END_FUNCTION
